(* IEC 61131-3 sources: TIA2AX/tests/V18/test_projects/expected/HW_2000482/6A1_AS10.2_AS11, 7 files *)

(* ---- HwIdentifiers.st ---- *)
TYPE
	HwIdentifiers : WORD
	(
		_6A1_AS10_2_AS11_Rail_0 :=	WORD#256,
		_6A1_AS10_2_AS11 :=	WORD#48,
		_6A1_AS10_2_AS11_Card_reader_writer_1 :=	WORD#51,
		_6A1_AS10_2_AS11_CPU_display_1 :=	WORD#54,
		_6A1_AS10_2_AS11_OPC_UA_1 :=	WORD#117,
		_6A1_AS10_2_AS11_PROFINET_interface_1 :=	WORD#64,
		_6A1_AS10_2_AS11_PROFINET_interface_1_Port_1 :=	WORD#65,
		_6A1_AS10_2_AS11_PROFINET_interface_1_Port_2 :=	WORD#66,
		_6A1_AS10_2_AS11_PROFINET_interface_2 :=	WORD#72,
		_6A1_AS10_2_AS11_PROFINET_interface_2_Port_1 :=	WORD#73,
		CPX_PneuOst_AS11_PN_IO_Interface :=	WORD#259,
		CPX_PneuOst_AS11_PN_IO_Interface_Port_1 :=	WORD#260,
		CPX_PneuOst_AS11_PN_IO_Interface_Port_2 :=	WORD#261,
		CPX_PneuOst_AS11_CPX :=	WORD#262,
		CPX_PneuOst_AS11_FB33_PNIO_Module_1 :=	WORD#263,
		CPX_PneuOst_AS11_MPA1S_VMPA1_FB_EMS_8_8DO_1 :=	WORD#264,
		CPX_PneuOst_AS11_MPA2S_VMPA2_FB_EMS_4_4DO_2 :=	WORD#265,
		CPX_PneuOst_AS11_MPA2S_VMPA2_FB_EMS_4_4DO_1 :=	WORD#266,
		CPX_PneuOst_AS11_MPA1S_VMPA1_FB_EMS_8_8DO_3 :=	WORD#267,
		CPX_PneuOst_AS11_MPA1S_VMPA1_FB_EMS_8_8DO_4 :=	WORD#268,
		CPX_PneuOst_AS11_MPA1G_VMPA1_FB_EMG_8_8DO_1 :=	WORD#269,
		_6A2_AS11_Rack_0 :=	WORD#273,
		_6A2_AS11 :=	WORD#274,
		_6A2_AS11_6A2_AS11 :=	WORD#275,
		_6A2_AS11_PROFINET_interface :=	WORD#276,
		_6A2_AS11_PROFINET_interface_Port_1 :=	WORD#278,
		_6A2_AS11_PROFINET_interface_Port_2 :=	WORD#277,
		_6A2_AS11_BA_2xRJ45 :=	WORD#278,
		_6A2_AS11_6A3 :=	WORD#279,
		_6A2_AS11_6A5 :=	WORD#280,
		_6A2_AS11_6A13 :=	WORD#281,
		_6A2_AS11_6A20 :=	WORD#282,
		_6A2_AS11_Server_module_1 :=	WORD#283,
		HousingReader_AS11_Rack :=	WORD#285,
		HousingReader_AS11 :=	WORD#286,
		HousingReader_AS11_Interface :=	WORD#287,
		HousingReader_AS11_Interface_Port_1 :=	WORD#288,
		HousingReader_AS11_SR_75X :=	WORD#289,
		HousingReader_AS11_Handshake_and_General_Error_Status_Bits_1 :=	WORD#290,
		HousingReader_AS11_BUSY_Status_Bits_1 :=	WORD#291,
		HousingReader_AS11_Completion_Status_Bits_1 :=	WORD#292,
		HousingReader_AS11_Error_Status_Bits_1 :=	WORD#293,
		HousingReader_AS11_Terminal_Status_Bits_1 :=	WORD#294,
		HousingReader_AS11_Unstable_Read_Status_Bits_1 :=	WORD#295,
		HousingReader_AS11_Matching_Level_and_Total_Evaluation_Grade_Status_1 :=	WORD#296,
		HousingReader_AS11_Operation_Result_Status_1 :=	WORD#297,
		HousingReader_AS11_Read_Data_128Byte_1 :=	WORD#298,
		HousingReader_AS11_Latch_and_Error_Clear_Control_Bits_1 :=	WORD#299,
		HousingReader_AS11_Operation_instruction_Control_Bits_1 :=	WORD#300,
		HousingReader_AS11_Completion_Clear_Control_Bits_1 :=	WORD#301,
		HousingReader_AS11_Parameter_Bank_Number_1 :=	WORD#302,
		HousingReader_AS11_User_Data_128Byte_1 :=	WORD#303,
		as13_lan_Rack :=	WORD#305,
		as13_lan :=	WORD#306,
		as13_lan_Interface :=	WORD#307,
		as13_lan_Interface_Port_1 :=	WORD#308,
		as13_lan_Interface_Port_2 :=	WORD#309,
		as13_lan_Communication :=	WORD#310,
		CPX_PneuOst_AS10_2_PN_IO_Interface :=	WORD#314,
		CPX_PneuOst_AS10_2_PN_IO_Interface_Port_1 :=	WORD#315,
		CPX_PneuOst_AS10_2_PN_IO_Interface_Port_2 :=	WORD#316,
		CPX_PneuOst_AS10_2_CPX :=	WORD#317,
		CPX_PneuOst_AS10_2_FB33_PNIO_Module_1 :=	WORD#318,
		CPX_PneuOst_AS10_2_MPA1S_VMPA1_FB_EMS_8_8DO_1 :=	WORD#319,
		CPX_PneuOst_AS10_2_MPA1S_VMPA1_FB_EMS_8_8DO_3 :=	WORD#320,
		CPX_PneuOst_AS10_2_MPA1S_VMPA1_FB_EMS_8_8DO_2 :=	WORD#321,
		CPX_PneuOst_AS10_2_MPA1G_VMPA1_FB_EMG_8_8DO_1 :=	WORD#322,
		FlashingReader_Rack :=	WORD#324,
		FlashingReader :=	WORD#325,
		FlashingReader_Interface :=	WORD#326,
		FlashingReader_Interface_Port_1 :=	WORD#327,
		FlashingReader_SR_75X :=	WORD#328,
		FlashingReader_Handshake_and_General_Error_Status_Bits_1 :=	WORD#329,
		FlashingReader_BUSY_Status_Bits_1 :=	WORD#330,
		FlashingReader_Completion_Status_Bits_1 :=	WORD#331,
		FlashingReader_Error_Status_Bits_1 :=	WORD#332,
		FlashingReader_Terminal_Status_Bits_1 :=	WORD#333,
		FlashingReader_Unstable_Read_Status_Bits_1 :=	WORD#334,
		FlashingReader_Matching_Level_and_Total_Evaluation_Grade_Status_1 :=	WORD#335,
		FlashingReader_Operation_Result_Status_1 :=	WORD#336,
		FlashingReader_Read_Data_128Byte_1 :=	WORD#337,
		FlashingReader_Latch_and_Error_Clear_Control_Bits_1 :=	WORD#338,
		FlashingReader_Operation_instruction_Control_Bits_1 :=	WORD#339,
		FlashingReader_Completion_Clear_Control_Bits_1 :=	WORD#340,
		FlashingReader_Parameter_Bank_Number_1 :=	WORD#341,
		FlashingReader_User_Data_128Byte_1 :=	WORD#342,
		AS10_2flashing_Interface1 :=	WORD#346,
		AS10_2flashing_Interface1_Port1 :=	WORD#347,
		AS10_2flashing_DF_Profinet_IO :=	WORD#348,
		AS10_2flashing_In_64_Byte_1 :=	WORD#349,
		AS10_2flashing_Out_64_Byte_1 :=	WORD#350,
		NONE:= WORD#0
	);
END_TYPE

(* ---- HwInputs.st ---- *)
TYPE
	HwInputs : STRUCT
		_6A2_AS11_6A3 AT %B0 : WORD;
		_6A2_AS11_6A13 AT %B19 : ARRAY[0..31] OF BYTE;
		HousingReader_AS11_Handshake_and_General_Error_Status_Bits_1 AT %B51 : BYTE;
		HousingReader_AS11_BUSY_Status_Bits_1 AT %B52 : BYTE;
		HousingReader_AS11_Completion_Status_Bits_1 AT %B53 : BYTE;
		HousingReader_AS11_Error_Status_Bits_1 AT %B54 : BYTE;
		HousingReader_AS11_Terminal_Status_Bits_1 AT %B55 : BYTE;
		HousingReader_AS11_Unstable_Read_Status_Bits_1 AT %B56 : BYTE;
		HousingReader_AS11_Matching_Level_and_Total_Evaluation_Grade_Status_1 AT %B57 : ARRAY[0..7] OF BYTE;
		HousingReader_AS11_Operation_Result_Status_1 AT %B65 : ARRAY[0..19] OF BYTE;
		HousingReader_AS11_Read_Data_128Byte_1 AT %B85 : ARRAY[0..135] OF BYTE;
		as13_lan_as13_lan AT %B221 : BYTE;
		FlashingReader_Handshake_and_General_Error_Status_Bits_1 AT %B222 : BYTE;
		FlashingReader_BUSY_Status_Bits_1 AT %B223 : BYTE;
		FlashingReader_Completion_Status_Bits_1 AT %B224 : BYTE;
		FlashingReader_Error_Status_Bits_1 AT %B225 : BYTE;
		FlashingReader_Terminal_Status_Bits_1 AT %B226 : BYTE;
		FlashingReader_Unstable_Read_Status_Bits_1 AT %B227 : BYTE;
		FlashingReader_Matching_Level_and_Total_Evaluation_Grade_Status_1 AT %B228 : ARRAY[0..7] OF BYTE;
		FlashingReader_Operation_Result_Status_1 AT %B236 : ARRAY[0..19] OF BYTE;
		FlashingReader_Read_Data_128Byte_1 AT %B256 : ARRAY[0..135] OF BYTE;
		AS10_2flashing_In_64_Byte_1 AT %B528 : ARRAY[0..63] OF BYTE;
	END_STRUCT;
END_TYPE

(* ---- HwOutputs.st ---- *)
TYPE
	HwOutputs : STRUCT
		CPX_PneuOst_AS11_MPA1S_VMPA1_FB_EMS_8_8DO_1 AT %B13 : BYTE;
		CPX_PneuOst_AS11_MPA2S_VMPA2_FB_EMS_4_4DO_2 AT %B183 : BYTE;
		CPX_PneuOst_AS11_MPA2S_VMPA2_FB_EMS_4_4DO_1 AT %B193 : BYTE;
		CPX_PneuOst_AS11_MPA1S_VMPA1_FB_EMS_8_8DO_3 AT %B184 : BYTE;
		CPX_PneuOst_AS11_MPA1S_VMPA1_FB_EMS_8_8DO_4 AT %B185 : BYTE;
		CPX_PneuOst_AS11_MPA1G_VMPA1_FB_EMG_8_8DO_1 AT %B186 : BYTE;
		_6A2_AS11_6A5 AT %B0 : WORD;
		_6A2_AS11_6A13 AT %B19 : ARRAY[0..31] OF BYTE;
		_6A2_AS11_6A20 AT %B328 : ARRAY[0..7] OF BYTE;
		HousingReader_AS11_Latch_and_Error_Clear_Control_Bits_1 AT %B6 : BYTE;
		HousingReader_AS11_Operation_instruction_Control_Bits_1 AT %B7 : BYTE;
		HousingReader_AS11_Completion_Clear_Control_Bits_1 AT %B12 : BYTE;
		HousingReader_AS11_Parameter_Bank_Number_1 AT %B51 : WORD;
		HousingReader_AS11_User_Data_128Byte_1 AT %B53 : ARRAY[0..129] OF BYTE;
		CPX_PneuOst_AS10_2_MPA1S_VMPA1_FB_EMS_8_8DO_1 AT %B188 : BYTE;
		CPX_PneuOst_AS10_2_MPA1S_VMPA1_FB_EMS_8_8DO_3 AT %B190 : BYTE;
		CPX_PneuOst_AS10_2_MPA1S_VMPA1_FB_EMS_8_8DO_2 AT %B194 : BYTE;
		CPX_PneuOst_AS10_2_MPA1G_VMPA1_FB_EMG_8_8DO_1 AT %B189 : BYTE;
		FlashingReader_Latch_and_Error_Clear_Control_Bits_1 AT %B191 : BYTE;
		FlashingReader_Operation_instruction_Control_Bits_1 AT %B192 : BYTE;
		FlashingReader_Completion_Clear_Control_Bits_1 AT %B195 : BYTE;
		FlashingReader_Parameter_Bank_Number_1 AT %B196 : WORD;
		FlashingReader_User_Data_128Byte_1 AT %B198 : ARRAY[0..129] OF BYTE;
		AS10_2flashing_Out_64_Byte_1 AT %B523 : ARRAY[0..63] OF BYTE;
	END_STRUCT;
END_TYPE

(* ---- PlcInputs.st ---- *)
TYPE
	PlcInputs : STRUCT
		_6A2_AS11_6A3 : WORD;
		_6A2_AS11_6A13 : ARRAY[0..31] OF BYTE;
		HousingReader_AS11_Handshake_and_General_Error_Status_Bits_1 : BYTE;
		HousingReader_AS11_BUSY_Status_Bits_1 : BYTE;
		HousingReader_AS11_Completion_Status_Bits_1 : BYTE;
		HousingReader_AS11_Error_Status_Bits_1 : BYTE;
		HousingReader_AS11_Terminal_Status_Bits_1 : BYTE;
		HousingReader_AS11_Unstable_Read_Status_Bits_1 : BYTE;
		HousingReader_AS11_Matching_Level_and_Total_Evaluation_Grade_Status_1 : ARRAY[0..7] OF BYTE;
		HousingReader_AS11_Operation_Result_Status_1 : ARRAY[0..19] OF BYTE;
		HousingReader_AS11_Read_Data_128Byte_1 : ARRAY[0..135] OF BYTE;
		as13_lan_as13_lan : BYTE;
		FlashingReader_Handshake_and_General_Error_Status_Bits_1 : BYTE;
		FlashingReader_BUSY_Status_Bits_1 : BYTE;
		FlashingReader_Completion_Status_Bits_1 : BYTE;
		FlashingReader_Error_Status_Bits_1 : BYTE;
		FlashingReader_Terminal_Status_Bits_1 : BYTE;
		FlashingReader_Unstable_Read_Status_Bits_1 : BYTE;
		FlashingReader_Matching_Level_and_Total_Evaluation_Grade_Status_1 : ARRAY[0..7] OF BYTE;
		FlashingReader_Operation_Result_Status_1 : ARRAY[0..19] OF BYTE;
		FlashingReader_Read_Data_128Byte_1 : ARRAY[0..135] OF BYTE;
		AS10_2flashing_In_64_Byte_1 : ARRAY[0..63] OF BYTE;
	END_STRUCT;
END_TYPE

(* ---- PlcOutputs.st ---- *)
TYPE
	PlcOutputs : STRUCT
		CPX_PneuOst_AS11_MPA1S_VMPA1_FB_EMS_8_8DO_1 : BYTE;
		CPX_PneuOst_AS11_MPA2S_VMPA2_FB_EMS_4_4DO_2 : BYTE;
		CPX_PneuOst_AS11_MPA2S_VMPA2_FB_EMS_4_4DO_1 : BYTE;
		CPX_PneuOst_AS11_MPA1S_VMPA1_FB_EMS_8_8DO_3 : BYTE;
		CPX_PneuOst_AS11_MPA1S_VMPA1_FB_EMS_8_8DO_4 : BYTE;
		CPX_PneuOst_AS11_MPA1G_VMPA1_FB_EMG_8_8DO_1 : BYTE;
		_6A2_AS11_6A5 : WORD;
		_6A2_AS11_6A13 : ARRAY[0..31] OF BYTE;
		_6A2_AS11_6A20 : ARRAY[0..7] OF BYTE;
		HousingReader_AS11_Latch_and_Error_Clear_Control_Bits_1 : BYTE;
		HousingReader_AS11_Operation_instruction_Control_Bits_1 : BYTE;
		HousingReader_AS11_Completion_Clear_Control_Bits_1 : BYTE;
		HousingReader_AS11_Parameter_Bank_Number_1 : WORD;
		HousingReader_AS11_User_Data_128Byte_1 : ARRAY[0..129] OF BYTE;
		CPX_PneuOst_AS10_2_MPA1S_VMPA1_FB_EMS_8_8DO_1 : BYTE;
		CPX_PneuOst_AS10_2_MPA1S_VMPA1_FB_EMS_8_8DO_3 : BYTE;
		CPX_PneuOst_AS10_2_MPA1S_VMPA1_FB_EMS_8_8DO_2 : BYTE;
		CPX_PneuOst_AS10_2_MPA1G_VMPA1_FB_EMG_8_8DO_1 : BYTE;
		FlashingReader_Latch_and_Error_Clear_Control_Bits_1 : BYTE;
		FlashingReader_Operation_instruction_Control_Bits_1 : BYTE;
		FlashingReader_Completion_Clear_Control_Bits_1 : BYTE;
		FlashingReader_Parameter_Bank_Number_1 : WORD;
		FlashingReader_User_Data_128Byte_1 : ARRAY[0..129] OF BYTE;
		AS10_2flashing_Out_64_Byte_1 : ARRAY[0..63] OF BYTE;
	END_STRUCT;
END_TYPE

(* ---- CopyInputs.st ---- *)
FUNCTION CopyInputs
	VAR_EXTERNAL
		HwInputs : HwInputs;
		PlcInputs : PlcInputs;
	END_VAR
	PlcInputs._6A2_AS11_6A3 := HwInputs._6A2_AS11_6A3;
	PlcInputs._6A2_AS11_6A13[0] := HwInputs._6A2_AS11_6A13[0];
	PlcInputs._6A2_AS11_6A13[1] := HwInputs._6A2_AS11_6A13[1];
	PlcInputs._6A2_AS11_6A13[2] := HwInputs._6A2_AS11_6A13[2];
	PlcInputs._6A2_AS11_6A13[3] := HwInputs._6A2_AS11_6A13[3];
	PlcInputs._6A2_AS11_6A13[4] := HwInputs._6A2_AS11_6A13[4];
	PlcInputs._6A2_AS11_6A13[5] := HwInputs._6A2_AS11_6A13[5];
	PlcInputs._6A2_AS11_6A13[6] := HwInputs._6A2_AS11_6A13[6];
	PlcInputs._6A2_AS11_6A13[7] := HwInputs._6A2_AS11_6A13[7];
	PlcInputs._6A2_AS11_6A13[8] := HwInputs._6A2_AS11_6A13[8];
	PlcInputs._6A2_AS11_6A13[9] := HwInputs._6A2_AS11_6A13[9];
	PlcInputs._6A2_AS11_6A13[10] := HwInputs._6A2_AS11_6A13[10];
	PlcInputs._6A2_AS11_6A13[11] := HwInputs._6A2_AS11_6A13[11];
	PlcInputs._6A2_AS11_6A13[12] := HwInputs._6A2_AS11_6A13[12];
	PlcInputs._6A2_AS11_6A13[13] := HwInputs._6A2_AS11_6A13[13];
	PlcInputs._6A2_AS11_6A13[14] := HwInputs._6A2_AS11_6A13[14];
	PlcInputs._6A2_AS11_6A13[15] := HwInputs._6A2_AS11_6A13[15];
	PlcInputs._6A2_AS11_6A13[16] := HwInputs._6A2_AS11_6A13[16];
	PlcInputs._6A2_AS11_6A13[17] := HwInputs._6A2_AS11_6A13[17];
	PlcInputs._6A2_AS11_6A13[18] := HwInputs._6A2_AS11_6A13[18];
	PlcInputs._6A2_AS11_6A13[19] := HwInputs._6A2_AS11_6A13[19];
	PlcInputs._6A2_AS11_6A13[20] := HwInputs._6A2_AS11_6A13[20];
	PlcInputs._6A2_AS11_6A13[21] := HwInputs._6A2_AS11_6A13[21];
	PlcInputs._6A2_AS11_6A13[22] := HwInputs._6A2_AS11_6A13[22];
	PlcInputs._6A2_AS11_6A13[23] := HwInputs._6A2_AS11_6A13[23];
	PlcInputs._6A2_AS11_6A13[24] := HwInputs._6A2_AS11_6A13[24];
	PlcInputs._6A2_AS11_6A13[25] := HwInputs._6A2_AS11_6A13[25];
	PlcInputs._6A2_AS11_6A13[26] := HwInputs._6A2_AS11_6A13[26];
	PlcInputs._6A2_AS11_6A13[27] := HwInputs._6A2_AS11_6A13[27];
	PlcInputs._6A2_AS11_6A13[28] := HwInputs._6A2_AS11_6A13[28];
	PlcInputs._6A2_AS11_6A13[29] := HwInputs._6A2_AS11_6A13[29];
	PlcInputs._6A2_AS11_6A13[30] := HwInputs._6A2_AS11_6A13[30];
	PlcInputs._6A2_AS11_6A13[31] := HwInputs._6A2_AS11_6A13[31];
	PlcInputs.HousingReader_AS11_Handshake_and_General_Error_Status_Bits_1 := HwInputs.HousingReader_AS11_Handshake_and_General_Error_Status_Bits_1;
	PlcInputs.HousingReader_AS11_BUSY_Status_Bits_1 := HwInputs.HousingReader_AS11_BUSY_Status_Bits_1;
	PlcInputs.HousingReader_AS11_Completion_Status_Bits_1 := HwInputs.HousingReader_AS11_Completion_Status_Bits_1;
	PlcInputs.HousingReader_AS11_Error_Status_Bits_1 := HwInputs.HousingReader_AS11_Error_Status_Bits_1;
	PlcInputs.HousingReader_AS11_Terminal_Status_Bits_1 := HwInputs.HousingReader_AS11_Terminal_Status_Bits_1;
	PlcInputs.HousingReader_AS11_Unstable_Read_Status_Bits_1 := HwInputs.HousingReader_AS11_Unstable_Read_Status_Bits_1;
	PlcInputs.HousingReader_AS11_Matching_Level_and_Total_Evaluation_Grade_Status_1[0] := HwInputs.HousingReader_AS11_Matching_Level_and_Total_Evaluation_Grade_Status_1[0];
	PlcInputs.HousingReader_AS11_Matching_Level_and_Total_Evaluation_Grade_Status_1[1] := HwInputs.HousingReader_AS11_Matching_Level_and_Total_Evaluation_Grade_Status_1[1];
	PlcInputs.HousingReader_AS11_Matching_Level_and_Total_Evaluation_Grade_Status_1[2] := HwInputs.HousingReader_AS11_Matching_Level_and_Total_Evaluation_Grade_Status_1[2];
	PlcInputs.HousingReader_AS11_Matching_Level_and_Total_Evaluation_Grade_Status_1[3] := HwInputs.HousingReader_AS11_Matching_Level_and_Total_Evaluation_Grade_Status_1[3];
	PlcInputs.HousingReader_AS11_Matching_Level_and_Total_Evaluation_Grade_Status_1[4] := HwInputs.HousingReader_AS11_Matching_Level_and_Total_Evaluation_Grade_Status_1[4];
	PlcInputs.HousingReader_AS11_Matching_Level_and_Total_Evaluation_Grade_Status_1[5] := HwInputs.HousingReader_AS11_Matching_Level_and_Total_Evaluation_Grade_Status_1[5];
	PlcInputs.HousingReader_AS11_Matching_Level_and_Total_Evaluation_Grade_Status_1[6] := HwInputs.HousingReader_AS11_Matching_Level_and_Total_Evaluation_Grade_Status_1[6];
	PlcInputs.HousingReader_AS11_Matching_Level_and_Total_Evaluation_Grade_Status_1[7] := HwInputs.HousingReader_AS11_Matching_Level_and_Total_Evaluation_Grade_Status_1[7];
	PlcInputs.HousingReader_AS11_Operation_Result_Status_1[0] := HwInputs.HousingReader_AS11_Operation_Result_Status_1[0];
	PlcInputs.HousingReader_AS11_Operation_Result_Status_1[1] := HwInputs.HousingReader_AS11_Operation_Result_Status_1[1];
	PlcInputs.HousingReader_AS11_Operation_Result_Status_1[2] := HwInputs.HousingReader_AS11_Operation_Result_Status_1[2];
	PlcInputs.HousingReader_AS11_Operation_Result_Status_1[3] := HwInputs.HousingReader_AS11_Operation_Result_Status_1[3];
	PlcInputs.HousingReader_AS11_Operation_Result_Status_1[4] := HwInputs.HousingReader_AS11_Operation_Result_Status_1[4];
	PlcInputs.HousingReader_AS11_Operation_Result_Status_1[5] := HwInputs.HousingReader_AS11_Operation_Result_Status_1[5];
	PlcInputs.HousingReader_AS11_Operation_Result_Status_1[6] := HwInputs.HousingReader_AS11_Operation_Result_Status_1[6];
	PlcInputs.HousingReader_AS11_Operation_Result_Status_1[7] := HwInputs.HousingReader_AS11_Operation_Result_Status_1[7];
	PlcInputs.HousingReader_AS11_Operation_Result_Status_1[8] := HwInputs.HousingReader_AS11_Operation_Result_Status_1[8];
	PlcInputs.HousingReader_AS11_Operation_Result_Status_1[9] := HwInputs.HousingReader_AS11_Operation_Result_Status_1[9];
	PlcInputs.HousingReader_AS11_Operation_Result_Status_1[10] := HwInputs.HousingReader_AS11_Operation_Result_Status_1[10];
	PlcInputs.HousingReader_AS11_Operation_Result_Status_1[11] := HwInputs.HousingReader_AS11_Operation_Result_Status_1[11];
	PlcInputs.HousingReader_AS11_Operation_Result_Status_1[12] := HwInputs.HousingReader_AS11_Operation_Result_Status_1[12];
	PlcInputs.HousingReader_AS11_Operation_Result_Status_1[13] := HwInputs.HousingReader_AS11_Operation_Result_Status_1[13];
	PlcInputs.HousingReader_AS11_Operation_Result_Status_1[14] := HwInputs.HousingReader_AS11_Operation_Result_Status_1[14];
	PlcInputs.HousingReader_AS11_Operation_Result_Status_1[15] := HwInputs.HousingReader_AS11_Operation_Result_Status_1[15];
	PlcInputs.HousingReader_AS11_Operation_Result_Status_1[16] := HwInputs.HousingReader_AS11_Operation_Result_Status_1[16];
	PlcInputs.HousingReader_AS11_Operation_Result_Status_1[17] := HwInputs.HousingReader_AS11_Operation_Result_Status_1[17];
	PlcInputs.HousingReader_AS11_Operation_Result_Status_1[18] := HwInputs.HousingReader_AS11_Operation_Result_Status_1[18];
	PlcInputs.HousingReader_AS11_Operation_Result_Status_1[19] := HwInputs.HousingReader_AS11_Operation_Result_Status_1[19];
	PlcInputs.HousingReader_AS11_Read_Data_128Byte_1[0] := HwInputs.HousingReader_AS11_Read_Data_128Byte_1[0];
	PlcInputs.HousingReader_AS11_Read_Data_128Byte_1[1] := HwInputs.HousingReader_AS11_Read_Data_128Byte_1[1];
	PlcInputs.HousingReader_AS11_Read_Data_128Byte_1[2] := HwInputs.HousingReader_AS11_Read_Data_128Byte_1[2];
	PlcInputs.HousingReader_AS11_Read_Data_128Byte_1[3] := HwInputs.HousingReader_AS11_Read_Data_128Byte_1[3];
	PlcInputs.HousingReader_AS11_Read_Data_128Byte_1[4] := HwInputs.HousingReader_AS11_Read_Data_128Byte_1[4];
	PlcInputs.HousingReader_AS11_Read_Data_128Byte_1[5] := HwInputs.HousingReader_AS11_Read_Data_128Byte_1[5];
	PlcInputs.HousingReader_AS11_Read_Data_128Byte_1[6] := HwInputs.HousingReader_AS11_Read_Data_128Byte_1[6];
	PlcInputs.HousingReader_AS11_Read_Data_128Byte_1[7] := HwInputs.HousingReader_AS11_Read_Data_128Byte_1[7];
	PlcInputs.HousingReader_AS11_Read_Data_128Byte_1[8] := HwInputs.HousingReader_AS11_Read_Data_128Byte_1[8];
	PlcInputs.HousingReader_AS11_Read_Data_128Byte_1[9] := HwInputs.HousingReader_AS11_Read_Data_128Byte_1[9];
	PlcInputs.HousingReader_AS11_Read_Data_128Byte_1[10] := HwInputs.HousingReader_AS11_Read_Data_128Byte_1[10];
	PlcInputs.HousingReader_AS11_Read_Data_128Byte_1[11] := HwInputs.HousingReader_AS11_Read_Data_128Byte_1[11];
	PlcInputs.HousingReader_AS11_Read_Data_128Byte_1[12] := HwInputs.HousingReader_AS11_Read_Data_128Byte_1[12];
	PlcInputs.HousingReader_AS11_Read_Data_128Byte_1[13] := HwInputs.HousingReader_AS11_Read_Data_128Byte_1[13];
	PlcInputs.HousingReader_AS11_Read_Data_128Byte_1[14] := HwInputs.HousingReader_AS11_Read_Data_128Byte_1[14];
	PlcInputs.HousingReader_AS11_Read_Data_128Byte_1[15] := HwInputs.HousingReader_AS11_Read_Data_128Byte_1[15];
	PlcInputs.HousingReader_AS11_Read_Data_128Byte_1[16] := HwInputs.HousingReader_AS11_Read_Data_128Byte_1[16];
	PlcInputs.HousingReader_AS11_Read_Data_128Byte_1[17] := HwInputs.HousingReader_AS11_Read_Data_128Byte_1[17];
	PlcInputs.HousingReader_AS11_Read_Data_128Byte_1[18] := HwInputs.HousingReader_AS11_Read_Data_128Byte_1[18];
	PlcInputs.HousingReader_AS11_Read_Data_128Byte_1[19] := HwInputs.HousingReader_AS11_Read_Data_128Byte_1[19];
	PlcInputs.HousingReader_AS11_Read_Data_128Byte_1[20] := HwInputs.HousingReader_AS11_Read_Data_128Byte_1[20];
	PlcInputs.HousingReader_AS11_Read_Data_128Byte_1[21] := HwInputs.HousingReader_AS11_Read_Data_128Byte_1[21];
	PlcInputs.HousingReader_AS11_Read_Data_128Byte_1[22] := HwInputs.HousingReader_AS11_Read_Data_128Byte_1[22];
	PlcInputs.HousingReader_AS11_Read_Data_128Byte_1[23] := HwInputs.HousingReader_AS11_Read_Data_128Byte_1[23];
	PlcInputs.HousingReader_AS11_Read_Data_128Byte_1[24] := HwInputs.HousingReader_AS11_Read_Data_128Byte_1[24];
	PlcInputs.HousingReader_AS11_Read_Data_128Byte_1[25] := HwInputs.HousingReader_AS11_Read_Data_128Byte_1[25];
	PlcInputs.HousingReader_AS11_Read_Data_128Byte_1[26] := HwInputs.HousingReader_AS11_Read_Data_128Byte_1[26];
	PlcInputs.HousingReader_AS11_Read_Data_128Byte_1[27] := HwInputs.HousingReader_AS11_Read_Data_128Byte_1[27];
	PlcInputs.HousingReader_AS11_Read_Data_128Byte_1[28] := HwInputs.HousingReader_AS11_Read_Data_128Byte_1[28];
	PlcInputs.HousingReader_AS11_Read_Data_128Byte_1[29] := HwInputs.HousingReader_AS11_Read_Data_128Byte_1[29];
	PlcInputs.HousingReader_AS11_Read_Data_128Byte_1[30] := HwInputs.HousingReader_AS11_Read_Data_128Byte_1[30];
	PlcInputs.HousingReader_AS11_Read_Data_128Byte_1[31] := HwInputs.HousingReader_AS11_Read_Data_128Byte_1[31];
	PlcInputs.HousingReader_AS11_Read_Data_128Byte_1[32] := HwInputs.HousingReader_AS11_Read_Data_128Byte_1[32];
	PlcInputs.HousingReader_AS11_Read_Data_128Byte_1[33] := HwInputs.HousingReader_AS11_Read_Data_128Byte_1[33];
	PlcInputs.HousingReader_AS11_Read_Data_128Byte_1[34] := HwInputs.HousingReader_AS11_Read_Data_128Byte_1[34];
	PlcInputs.HousingReader_AS11_Read_Data_128Byte_1[35] := HwInputs.HousingReader_AS11_Read_Data_128Byte_1[35];
	PlcInputs.HousingReader_AS11_Read_Data_128Byte_1[36] := HwInputs.HousingReader_AS11_Read_Data_128Byte_1[36];
	PlcInputs.HousingReader_AS11_Read_Data_128Byte_1[37] := HwInputs.HousingReader_AS11_Read_Data_128Byte_1[37];
	PlcInputs.HousingReader_AS11_Read_Data_128Byte_1[38] := HwInputs.HousingReader_AS11_Read_Data_128Byte_1[38];
	PlcInputs.HousingReader_AS11_Read_Data_128Byte_1[39] := HwInputs.HousingReader_AS11_Read_Data_128Byte_1[39];
	PlcInputs.HousingReader_AS11_Read_Data_128Byte_1[40] := HwInputs.HousingReader_AS11_Read_Data_128Byte_1[40];
	PlcInputs.HousingReader_AS11_Read_Data_128Byte_1[41] := HwInputs.HousingReader_AS11_Read_Data_128Byte_1[41];
	PlcInputs.HousingReader_AS11_Read_Data_128Byte_1[42] := HwInputs.HousingReader_AS11_Read_Data_128Byte_1[42];
	PlcInputs.HousingReader_AS11_Read_Data_128Byte_1[43] := HwInputs.HousingReader_AS11_Read_Data_128Byte_1[43];
	PlcInputs.HousingReader_AS11_Read_Data_128Byte_1[44] := HwInputs.HousingReader_AS11_Read_Data_128Byte_1[44];
	PlcInputs.HousingReader_AS11_Read_Data_128Byte_1[45] := HwInputs.HousingReader_AS11_Read_Data_128Byte_1[45];
	PlcInputs.HousingReader_AS11_Read_Data_128Byte_1[46] := HwInputs.HousingReader_AS11_Read_Data_128Byte_1[46];
	PlcInputs.HousingReader_AS11_Read_Data_128Byte_1[47] := HwInputs.HousingReader_AS11_Read_Data_128Byte_1[47];
	PlcInputs.HousingReader_AS11_Read_Data_128Byte_1[48] := HwInputs.HousingReader_AS11_Read_Data_128Byte_1[48];
	PlcInputs.HousingReader_AS11_Read_Data_128Byte_1[49] := HwInputs.HousingReader_AS11_Read_Data_128Byte_1[49];
	PlcInputs.HousingReader_AS11_Read_Data_128Byte_1[50] := HwInputs.HousingReader_AS11_Read_Data_128Byte_1[50];
	PlcInputs.HousingReader_AS11_Read_Data_128Byte_1[51] := HwInputs.HousingReader_AS11_Read_Data_128Byte_1[51];
	PlcInputs.HousingReader_AS11_Read_Data_128Byte_1[52] := HwInputs.HousingReader_AS11_Read_Data_128Byte_1[52];
	PlcInputs.HousingReader_AS11_Read_Data_128Byte_1[53] := HwInputs.HousingReader_AS11_Read_Data_128Byte_1[53];
	PlcInputs.HousingReader_AS11_Read_Data_128Byte_1[54] := HwInputs.HousingReader_AS11_Read_Data_128Byte_1[54];
	PlcInputs.HousingReader_AS11_Read_Data_128Byte_1[55] := HwInputs.HousingReader_AS11_Read_Data_128Byte_1[55];
	PlcInputs.HousingReader_AS11_Read_Data_128Byte_1[56] := HwInputs.HousingReader_AS11_Read_Data_128Byte_1[56];
	PlcInputs.HousingReader_AS11_Read_Data_128Byte_1[57] := HwInputs.HousingReader_AS11_Read_Data_128Byte_1[57];
	PlcInputs.HousingReader_AS11_Read_Data_128Byte_1[58] := HwInputs.HousingReader_AS11_Read_Data_128Byte_1[58];
	PlcInputs.HousingReader_AS11_Read_Data_128Byte_1[59] := HwInputs.HousingReader_AS11_Read_Data_128Byte_1[59];
	PlcInputs.HousingReader_AS11_Read_Data_128Byte_1[60] := HwInputs.HousingReader_AS11_Read_Data_128Byte_1[60];
	PlcInputs.HousingReader_AS11_Read_Data_128Byte_1[61] := HwInputs.HousingReader_AS11_Read_Data_128Byte_1[61];
	PlcInputs.HousingReader_AS11_Read_Data_128Byte_1[62] := HwInputs.HousingReader_AS11_Read_Data_128Byte_1[62];
	PlcInputs.HousingReader_AS11_Read_Data_128Byte_1[63] := HwInputs.HousingReader_AS11_Read_Data_128Byte_1[63];
	PlcInputs.HousingReader_AS11_Read_Data_128Byte_1[64] := HwInputs.HousingReader_AS11_Read_Data_128Byte_1[64];
	PlcInputs.HousingReader_AS11_Read_Data_128Byte_1[65] := HwInputs.HousingReader_AS11_Read_Data_128Byte_1[65];
	PlcInputs.HousingReader_AS11_Read_Data_128Byte_1[66] := HwInputs.HousingReader_AS11_Read_Data_128Byte_1[66];
	PlcInputs.HousingReader_AS11_Read_Data_128Byte_1[67] := HwInputs.HousingReader_AS11_Read_Data_128Byte_1[67];
	PlcInputs.HousingReader_AS11_Read_Data_128Byte_1[68] := HwInputs.HousingReader_AS11_Read_Data_128Byte_1[68];
	PlcInputs.HousingReader_AS11_Read_Data_128Byte_1[69] := HwInputs.HousingReader_AS11_Read_Data_128Byte_1[69];
	PlcInputs.HousingReader_AS11_Read_Data_128Byte_1[70] := HwInputs.HousingReader_AS11_Read_Data_128Byte_1[70];
	PlcInputs.HousingReader_AS11_Read_Data_128Byte_1[71] := HwInputs.HousingReader_AS11_Read_Data_128Byte_1[71];
	PlcInputs.HousingReader_AS11_Read_Data_128Byte_1[72] := HwInputs.HousingReader_AS11_Read_Data_128Byte_1[72];
	PlcInputs.HousingReader_AS11_Read_Data_128Byte_1[73] := HwInputs.HousingReader_AS11_Read_Data_128Byte_1[73];
	PlcInputs.HousingReader_AS11_Read_Data_128Byte_1[74] := HwInputs.HousingReader_AS11_Read_Data_128Byte_1[74];
	PlcInputs.HousingReader_AS11_Read_Data_128Byte_1[75] := HwInputs.HousingReader_AS11_Read_Data_128Byte_1[75];
	PlcInputs.HousingReader_AS11_Read_Data_128Byte_1[76] := HwInputs.HousingReader_AS11_Read_Data_128Byte_1[76];
	PlcInputs.HousingReader_AS11_Read_Data_128Byte_1[77] := HwInputs.HousingReader_AS11_Read_Data_128Byte_1[77];
	PlcInputs.HousingReader_AS11_Read_Data_128Byte_1[78] := HwInputs.HousingReader_AS11_Read_Data_128Byte_1[78];
	PlcInputs.HousingReader_AS11_Read_Data_128Byte_1[79] := HwInputs.HousingReader_AS11_Read_Data_128Byte_1[79];
	PlcInputs.HousingReader_AS11_Read_Data_128Byte_1[80] := HwInputs.HousingReader_AS11_Read_Data_128Byte_1[80];
	PlcInputs.HousingReader_AS11_Read_Data_128Byte_1[81] := HwInputs.HousingReader_AS11_Read_Data_128Byte_1[81];
	PlcInputs.HousingReader_AS11_Read_Data_128Byte_1[82] := HwInputs.HousingReader_AS11_Read_Data_128Byte_1[82];
	PlcInputs.HousingReader_AS11_Read_Data_128Byte_1[83] := HwInputs.HousingReader_AS11_Read_Data_128Byte_1[83];
	PlcInputs.HousingReader_AS11_Read_Data_128Byte_1[84] := HwInputs.HousingReader_AS11_Read_Data_128Byte_1[84];
	PlcInputs.HousingReader_AS11_Read_Data_128Byte_1[85] := HwInputs.HousingReader_AS11_Read_Data_128Byte_1[85];
	PlcInputs.HousingReader_AS11_Read_Data_128Byte_1[86] := HwInputs.HousingReader_AS11_Read_Data_128Byte_1[86];
	PlcInputs.HousingReader_AS11_Read_Data_128Byte_1[87] := HwInputs.HousingReader_AS11_Read_Data_128Byte_1[87];
	PlcInputs.HousingReader_AS11_Read_Data_128Byte_1[88] := HwInputs.HousingReader_AS11_Read_Data_128Byte_1[88];
	PlcInputs.HousingReader_AS11_Read_Data_128Byte_1[89] := HwInputs.HousingReader_AS11_Read_Data_128Byte_1[89];
	PlcInputs.HousingReader_AS11_Read_Data_128Byte_1[90] := HwInputs.HousingReader_AS11_Read_Data_128Byte_1[90];
	PlcInputs.HousingReader_AS11_Read_Data_128Byte_1[91] := HwInputs.HousingReader_AS11_Read_Data_128Byte_1[91];
	PlcInputs.HousingReader_AS11_Read_Data_128Byte_1[92] := HwInputs.HousingReader_AS11_Read_Data_128Byte_1[92];
	PlcInputs.HousingReader_AS11_Read_Data_128Byte_1[93] := HwInputs.HousingReader_AS11_Read_Data_128Byte_1[93];
	PlcInputs.HousingReader_AS11_Read_Data_128Byte_1[94] := HwInputs.HousingReader_AS11_Read_Data_128Byte_1[94];
	PlcInputs.HousingReader_AS11_Read_Data_128Byte_1[95] := HwInputs.HousingReader_AS11_Read_Data_128Byte_1[95];
	PlcInputs.HousingReader_AS11_Read_Data_128Byte_1[96] := HwInputs.HousingReader_AS11_Read_Data_128Byte_1[96];
	PlcInputs.HousingReader_AS11_Read_Data_128Byte_1[97] := HwInputs.HousingReader_AS11_Read_Data_128Byte_1[97];
	PlcInputs.HousingReader_AS11_Read_Data_128Byte_1[98] := HwInputs.HousingReader_AS11_Read_Data_128Byte_1[98];
	PlcInputs.HousingReader_AS11_Read_Data_128Byte_1[99] := HwInputs.HousingReader_AS11_Read_Data_128Byte_1[99];
	PlcInputs.HousingReader_AS11_Read_Data_128Byte_1[100] := HwInputs.HousingReader_AS11_Read_Data_128Byte_1[100];
	PlcInputs.HousingReader_AS11_Read_Data_128Byte_1[101] := HwInputs.HousingReader_AS11_Read_Data_128Byte_1[101];
	PlcInputs.HousingReader_AS11_Read_Data_128Byte_1[102] := HwInputs.HousingReader_AS11_Read_Data_128Byte_1[102];
	PlcInputs.HousingReader_AS11_Read_Data_128Byte_1[103] := HwInputs.HousingReader_AS11_Read_Data_128Byte_1[103];
	PlcInputs.HousingReader_AS11_Read_Data_128Byte_1[104] := HwInputs.HousingReader_AS11_Read_Data_128Byte_1[104];
	PlcInputs.HousingReader_AS11_Read_Data_128Byte_1[105] := HwInputs.HousingReader_AS11_Read_Data_128Byte_1[105];
	PlcInputs.HousingReader_AS11_Read_Data_128Byte_1[106] := HwInputs.HousingReader_AS11_Read_Data_128Byte_1[106];
	PlcInputs.HousingReader_AS11_Read_Data_128Byte_1[107] := HwInputs.HousingReader_AS11_Read_Data_128Byte_1[107];
	PlcInputs.HousingReader_AS11_Read_Data_128Byte_1[108] := HwInputs.HousingReader_AS11_Read_Data_128Byte_1[108];
	PlcInputs.HousingReader_AS11_Read_Data_128Byte_1[109] := HwInputs.HousingReader_AS11_Read_Data_128Byte_1[109];
	PlcInputs.HousingReader_AS11_Read_Data_128Byte_1[110] := HwInputs.HousingReader_AS11_Read_Data_128Byte_1[110];
	PlcInputs.HousingReader_AS11_Read_Data_128Byte_1[111] := HwInputs.HousingReader_AS11_Read_Data_128Byte_1[111];
	PlcInputs.HousingReader_AS11_Read_Data_128Byte_1[112] := HwInputs.HousingReader_AS11_Read_Data_128Byte_1[112];
	PlcInputs.HousingReader_AS11_Read_Data_128Byte_1[113] := HwInputs.HousingReader_AS11_Read_Data_128Byte_1[113];
	PlcInputs.HousingReader_AS11_Read_Data_128Byte_1[114] := HwInputs.HousingReader_AS11_Read_Data_128Byte_1[114];
	PlcInputs.HousingReader_AS11_Read_Data_128Byte_1[115] := HwInputs.HousingReader_AS11_Read_Data_128Byte_1[115];
	PlcInputs.HousingReader_AS11_Read_Data_128Byte_1[116] := HwInputs.HousingReader_AS11_Read_Data_128Byte_1[116];
	PlcInputs.HousingReader_AS11_Read_Data_128Byte_1[117] := HwInputs.HousingReader_AS11_Read_Data_128Byte_1[117];
	PlcInputs.HousingReader_AS11_Read_Data_128Byte_1[118] := HwInputs.HousingReader_AS11_Read_Data_128Byte_1[118];
	PlcInputs.HousingReader_AS11_Read_Data_128Byte_1[119] := HwInputs.HousingReader_AS11_Read_Data_128Byte_1[119];
	PlcInputs.HousingReader_AS11_Read_Data_128Byte_1[120] := HwInputs.HousingReader_AS11_Read_Data_128Byte_1[120];
	PlcInputs.HousingReader_AS11_Read_Data_128Byte_1[121] := HwInputs.HousingReader_AS11_Read_Data_128Byte_1[121];
	PlcInputs.HousingReader_AS11_Read_Data_128Byte_1[122] := HwInputs.HousingReader_AS11_Read_Data_128Byte_1[122];
	PlcInputs.HousingReader_AS11_Read_Data_128Byte_1[123] := HwInputs.HousingReader_AS11_Read_Data_128Byte_1[123];
	PlcInputs.HousingReader_AS11_Read_Data_128Byte_1[124] := HwInputs.HousingReader_AS11_Read_Data_128Byte_1[124];
	PlcInputs.HousingReader_AS11_Read_Data_128Byte_1[125] := HwInputs.HousingReader_AS11_Read_Data_128Byte_1[125];
	PlcInputs.HousingReader_AS11_Read_Data_128Byte_1[126] := HwInputs.HousingReader_AS11_Read_Data_128Byte_1[126];
	PlcInputs.HousingReader_AS11_Read_Data_128Byte_1[127] := HwInputs.HousingReader_AS11_Read_Data_128Byte_1[127];
	PlcInputs.HousingReader_AS11_Read_Data_128Byte_1[128] := HwInputs.HousingReader_AS11_Read_Data_128Byte_1[128];
	PlcInputs.HousingReader_AS11_Read_Data_128Byte_1[129] := HwInputs.HousingReader_AS11_Read_Data_128Byte_1[129];
	PlcInputs.HousingReader_AS11_Read_Data_128Byte_1[130] := HwInputs.HousingReader_AS11_Read_Data_128Byte_1[130];
	PlcInputs.HousingReader_AS11_Read_Data_128Byte_1[131] := HwInputs.HousingReader_AS11_Read_Data_128Byte_1[131];
	PlcInputs.HousingReader_AS11_Read_Data_128Byte_1[132] := HwInputs.HousingReader_AS11_Read_Data_128Byte_1[132];
	PlcInputs.HousingReader_AS11_Read_Data_128Byte_1[133] := HwInputs.HousingReader_AS11_Read_Data_128Byte_1[133];
	PlcInputs.HousingReader_AS11_Read_Data_128Byte_1[134] := HwInputs.HousingReader_AS11_Read_Data_128Byte_1[134];
	PlcInputs.HousingReader_AS11_Read_Data_128Byte_1[135] := HwInputs.HousingReader_AS11_Read_Data_128Byte_1[135];
	PlcInputs.as13_lan_as13_lan := HwInputs.as13_lan_as13_lan;
	PlcInputs.FlashingReader_Handshake_and_General_Error_Status_Bits_1 := HwInputs.FlashingReader_Handshake_and_General_Error_Status_Bits_1;
	PlcInputs.FlashingReader_BUSY_Status_Bits_1 := HwInputs.FlashingReader_BUSY_Status_Bits_1;
	PlcInputs.FlashingReader_Completion_Status_Bits_1 := HwInputs.FlashingReader_Completion_Status_Bits_1;
	PlcInputs.FlashingReader_Error_Status_Bits_1 := HwInputs.FlashingReader_Error_Status_Bits_1;
	PlcInputs.FlashingReader_Terminal_Status_Bits_1 := HwInputs.FlashingReader_Terminal_Status_Bits_1;
	PlcInputs.FlashingReader_Unstable_Read_Status_Bits_1 := HwInputs.FlashingReader_Unstable_Read_Status_Bits_1;
	PlcInputs.FlashingReader_Matching_Level_and_Total_Evaluation_Grade_Status_1[0] := HwInputs.FlashingReader_Matching_Level_and_Total_Evaluation_Grade_Status_1[0];
	PlcInputs.FlashingReader_Matching_Level_and_Total_Evaluation_Grade_Status_1[1] := HwInputs.FlashingReader_Matching_Level_and_Total_Evaluation_Grade_Status_1[1];
	PlcInputs.FlashingReader_Matching_Level_and_Total_Evaluation_Grade_Status_1[2] := HwInputs.FlashingReader_Matching_Level_and_Total_Evaluation_Grade_Status_1[2];
	PlcInputs.FlashingReader_Matching_Level_and_Total_Evaluation_Grade_Status_1[3] := HwInputs.FlashingReader_Matching_Level_and_Total_Evaluation_Grade_Status_1[3];
	PlcInputs.FlashingReader_Matching_Level_and_Total_Evaluation_Grade_Status_1[4] := HwInputs.FlashingReader_Matching_Level_and_Total_Evaluation_Grade_Status_1[4];
	PlcInputs.FlashingReader_Matching_Level_and_Total_Evaluation_Grade_Status_1[5] := HwInputs.FlashingReader_Matching_Level_and_Total_Evaluation_Grade_Status_1[5];
	PlcInputs.FlashingReader_Matching_Level_and_Total_Evaluation_Grade_Status_1[6] := HwInputs.FlashingReader_Matching_Level_and_Total_Evaluation_Grade_Status_1[6];
	PlcInputs.FlashingReader_Matching_Level_and_Total_Evaluation_Grade_Status_1[7] := HwInputs.FlashingReader_Matching_Level_and_Total_Evaluation_Grade_Status_1[7];
	PlcInputs.FlashingReader_Operation_Result_Status_1[0] := HwInputs.FlashingReader_Operation_Result_Status_1[0];
	PlcInputs.FlashingReader_Operation_Result_Status_1[1] := HwInputs.FlashingReader_Operation_Result_Status_1[1];
	PlcInputs.FlashingReader_Operation_Result_Status_1[2] := HwInputs.FlashingReader_Operation_Result_Status_1[2];
	PlcInputs.FlashingReader_Operation_Result_Status_1[3] := HwInputs.FlashingReader_Operation_Result_Status_1[3];
	PlcInputs.FlashingReader_Operation_Result_Status_1[4] := HwInputs.FlashingReader_Operation_Result_Status_1[4];
	PlcInputs.FlashingReader_Operation_Result_Status_1[5] := HwInputs.FlashingReader_Operation_Result_Status_1[5];
	PlcInputs.FlashingReader_Operation_Result_Status_1[6] := HwInputs.FlashingReader_Operation_Result_Status_1[6];
	PlcInputs.FlashingReader_Operation_Result_Status_1[7] := HwInputs.FlashingReader_Operation_Result_Status_1[7];
	PlcInputs.FlashingReader_Operation_Result_Status_1[8] := HwInputs.FlashingReader_Operation_Result_Status_1[8];
	PlcInputs.FlashingReader_Operation_Result_Status_1[9] := HwInputs.FlashingReader_Operation_Result_Status_1[9];
	PlcInputs.FlashingReader_Operation_Result_Status_1[10] := HwInputs.FlashingReader_Operation_Result_Status_1[10];
	PlcInputs.FlashingReader_Operation_Result_Status_1[11] := HwInputs.FlashingReader_Operation_Result_Status_1[11];
	PlcInputs.FlashingReader_Operation_Result_Status_1[12] := HwInputs.FlashingReader_Operation_Result_Status_1[12];
	PlcInputs.FlashingReader_Operation_Result_Status_1[13] := HwInputs.FlashingReader_Operation_Result_Status_1[13];
	PlcInputs.FlashingReader_Operation_Result_Status_1[14] := HwInputs.FlashingReader_Operation_Result_Status_1[14];
	PlcInputs.FlashingReader_Operation_Result_Status_1[15] := HwInputs.FlashingReader_Operation_Result_Status_1[15];
	PlcInputs.FlashingReader_Operation_Result_Status_1[16] := HwInputs.FlashingReader_Operation_Result_Status_1[16];
	PlcInputs.FlashingReader_Operation_Result_Status_1[17] := HwInputs.FlashingReader_Operation_Result_Status_1[17];
	PlcInputs.FlashingReader_Operation_Result_Status_1[18] := HwInputs.FlashingReader_Operation_Result_Status_1[18];
	PlcInputs.FlashingReader_Operation_Result_Status_1[19] := HwInputs.FlashingReader_Operation_Result_Status_1[19];
	PlcInputs.FlashingReader_Read_Data_128Byte_1[0] := HwInputs.FlashingReader_Read_Data_128Byte_1[0];
	PlcInputs.FlashingReader_Read_Data_128Byte_1[1] := HwInputs.FlashingReader_Read_Data_128Byte_1[1];
	PlcInputs.FlashingReader_Read_Data_128Byte_1[2] := HwInputs.FlashingReader_Read_Data_128Byte_1[2];
	PlcInputs.FlashingReader_Read_Data_128Byte_1[3] := HwInputs.FlashingReader_Read_Data_128Byte_1[3];
	PlcInputs.FlashingReader_Read_Data_128Byte_1[4] := HwInputs.FlashingReader_Read_Data_128Byte_1[4];
	PlcInputs.FlashingReader_Read_Data_128Byte_1[5] := HwInputs.FlashingReader_Read_Data_128Byte_1[5];
	PlcInputs.FlashingReader_Read_Data_128Byte_1[6] := HwInputs.FlashingReader_Read_Data_128Byte_1[6];
	PlcInputs.FlashingReader_Read_Data_128Byte_1[7] := HwInputs.FlashingReader_Read_Data_128Byte_1[7];
	PlcInputs.FlashingReader_Read_Data_128Byte_1[8] := HwInputs.FlashingReader_Read_Data_128Byte_1[8];
	PlcInputs.FlashingReader_Read_Data_128Byte_1[9] := HwInputs.FlashingReader_Read_Data_128Byte_1[9];
	PlcInputs.FlashingReader_Read_Data_128Byte_1[10] := HwInputs.FlashingReader_Read_Data_128Byte_1[10];
	PlcInputs.FlashingReader_Read_Data_128Byte_1[11] := HwInputs.FlashingReader_Read_Data_128Byte_1[11];
	PlcInputs.FlashingReader_Read_Data_128Byte_1[12] := HwInputs.FlashingReader_Read_Data_128Byte_1[12];
	PlcInputs.FlashingReader_Read_Data_128Byte_1[13] := HwInputs.FlashingReader_Read_Data_128Byte_1[13];
	PlcInputs.FlashingReader_Read_Data_128Byte_1[14] := HwInputs.FlashingReader_Read_Data_128Byte_1[14];
	PlcInputs.FlashingReader_Read_Data_128Byte_1[15] := HwInputs.FlashingReader_Read_Data_128Byte_1[15];
	PlcInputs.FlashingReader_Read_Data_128Byte_1[16] := HwInputs.FlashingReader_Read_Data_128Byte_1[16];
	PlcInputs.FlashingReader_Read_Data_128Byte_1[17] := HwInputs.FlashingReader_Read_Data_128Byte_1[17];
	PlcInputs.FlashingReader_Read_Data_128Byte_1[18] := HwInputs.FlashingReader_Read_Data_128Byte_1[18];
	PlcInputs.FlashingReader_Read_Data_128Byte_1[19] := HwInputs.FlashingReader_Read_Data_128Byte_1[19];
	PlcInputs.FlashingReader_Read_Data_128Byte_1[20] := HwInputs.FlashingReader_Read_Data_128Byte_1[20];
	PlcInputs.FlashingReader_Read_Data_128Byte_1[21] := HwInputs.FlashingReader_Read_Data_128Byte_1[21];
	PlcInputs.FlashingReader_Read_Data_128Byte_1[22] := HwInputs.FlashingReader_Read_Data_128Byte_1[22];
	PlcInputs.FlashingReader_Read_Data_128Byte_1[23] := HwInputs.FlashingReader_Read_Data_128Byte_1[23];
	PlcInputs.FlashingReader_Read_Data_128Byte_1[24] := HwInputs.FlashingReader_Read_Data_128Byte_1[24];
	PlcInputs.FlashingReader_Read_Data_128Byte_1[25] := HwInputs.FlashingReader_Read_Data_128Byte_1[25];
	PlcInputs.FlashingReader_Read_Data_128Byte_1[26] := HwInputs.FlashingReader_Read_Data_128Byte_1[26];
	PlcInputs.FlashingReader_Read_Data_128Byte_1[27] := HwInputs.FlashingReader_Read_Data_128Byte_1[27];
	PlcInputs.FlashingReader_Read_Data_128Byte_1[28] := HwInputs.FlashingReader_Read_Data_128Byte_1[28];
	PlcInputs.FlashingReader_Read_Data_128Byte_1[29] := HwInputs.FlashingReader_Read_Data_128Byte_1[29];
	PlcInputs.FlashingReader_Read_Data_128Byte_1[30] := HwInputs.FlashingReader_Read_Data_128Byte_1[30];
	PlcInputs.FlashingReader_Read_Data_128Byte_1[31] := HwInputs.FlashingReader_Read_Data_128Byte_1[31];
	PlcInputs.FlashingReader_Read_Data_128Byte_1[32] := HwInputs.FlashingReader_Read_Data_128Byte_1[32];
	PlcInputs.FlashingReader_Read_Data_128Byte_1[33] := HwInputs.FlashingReader_Read_Data_128Byte_1[33];
	PlcInputs.FlashingReader_Read_Data_128Byte_1[34] := HwInputs.FlashingReader_Read_Data_128Byte_1[34];
	PlcInputs.FlashingReader_Read_Data_128Byte_1[35] := HwInputs.FlashingReader_Read_Data_128Byte_1[35];
	PlcInputs.FlashingReader_Read_Data_128Byte_1[36] := HwInputs.FlashingReader_Read_Data_128Byte_1[36];
	PlcInputs.FlashingReader_Read_Data_128Byte_1[37] := HwInputs.FlashingReader_Read_Data_128Byte_1[37];
	PlcInputs.FlashingReader_Read_Data_128Byte_1[38] := HwInputs.FlashingReader_Read_Data_128Byte_1[38];
	PlcInputs.FlashingReader_Read_Data_128Byte_1[39] := HwInputs.FlashingReader_Read_Data_128Byte_1[39];
	PlcInputs.FlashingReader_Read_Data_128Byte_1[40] := HwInputs.FlashingReader_Read_Data_128Byte_1[40];
	PlcInputs.FlashingReader_Read_Data_128Byte_1[41] := HwInputs.FlashingReader_Read_Data_128Byte_1[41];
	PlcInputs.FlashingReader_Read_Data_128Byte_1[42] := HwInputs.FlashingReader_Read_Data_128Byte_1[42];
	PlcInputs.FlashingReader_Read_Data_128Byte_1[43] := HwInputs.FlashingReader_Read_Data_128Byte_1[43];
	PlcInputs.FlashingReader_Read_Data_128Byte_1[44] := HwInputs.FlashingReader_Read_Data_128Byte_1[44];
	PlcInputs.FlashingReader_Read_Data_128Byte_1[45] := HwInputs.FlashingReader_Read_Data_128Byte_1[45];
	PlcInputs.FlashingReader_Read_Data_128Byte_1[46] := HwInputs.FlashingReader_Read_Data_128Byte_1[46];
	PlcInputs.FlashingReader_Read_Data_128Byte_1[47] := HwInputs.FlashingReader_Read_Data_128Byte_1[47];
	PlcInputs.FlashingReader_Read_Data_128Byte_1[48] := HwInputs.FlashingReader_Read_Data_128Byte_1[48];
	PlcInputs.FlashingReader_Read_Data_128Byte_1[49] := HwInputs.FlashingReader_Read_Data_128Byte_1[49];
	PlcInputs.FlashingReader_Read_Data_128Byte_1[50] := HwInputs.FlashingReader_Read_Data_128Byte_1[50];
	PlcInputs.FlashingReader_Read_Data_128Byte_1[51] := HwInputs.FlashingReader_Read_Data_128Byte_1[51];
	PlcInputs.FlashingReader_Read_Data_128Byte_1[52] := HwInputs.FlashingReader_Read_Data_128Byte_1[52];
	PlcInputs.FlashingReader_Read_Data_128Byte_1[53] := HwInputs.FlashingReader_Read_Data_128Byte_1[53];
	PlcInputs.FlashingReader_Read_Data_128Byte_1[54] := HwInputs.FlashingReader_Read_Data_128Byte_1[54];
	PlcInputs.FlashingReader_Read_Data_128Byte_1[55] := HwInputs.FlashingReader_Read_Data_128Byte_1[55];
	PlcInputs.FlashingReader_Read_Data_128Byte_1[56] := HwInputs.FlashingReader_Read_Data_128Byte_1[56];
	PlcInputs.FlashingReader_Read_Data_128Byte_1[57] := HwInputs.FlashingReader_Read_Data_128Byte_1[57];
	PlcInputs.FlashingReader_Read_Data_128Byte_1[58] := HwInputs.FlashingReader_Read_Data_128Byte_1[58];
	PlcInputs.FlashingReader_Read_Data_128Byte_1[59] := HwInputs.FlashingReader_Read_Data_128Byte_1[59];
	PlcInputs.FlashingReader_Read_Data_128Byte_1[60] := HwInputs.FlashingReader_Read_Data_128Byte_1[60];
	PlcInputs.FlashingReader_Read_Data_128Byte_1[61] := HwInputs.FlashingReader_Read_Data_128Byte_1[61];
	PlcInputs.FlashingReader_Read_Data_128Byte_1[62] := HwInputs.FlashingReader_Read_Data_128Byte_1[62];
	PlcInputs.FlashingReader_Read_Data_128Byte_1[63] := HwInputs.FlashingReader_Read_Data_128Byte_1[63];
	PlcInputs.FlashingReader_Read_Data_128Byte_1[64] := HwInputs.FlashingReader_Read_Data_128Byte_1[64];
	PlcInputs.FlashingReader_Read_Data_128Byte_1[65] := HwInputs.FlashingReader_Read_Data_128Byte_1[65];
	PlcInputs.FlashingReader_Read_Data_128Byte_1[66] := HwInputs.FlashingReader_Read_Data_128Byte_1[66];
	PlcInputs.FlashingReader_Read_Data_128Byte_1[67] := HwInputs.FlashingReader_Read_Data_128Byte_1[67];
	PlcInputs.FlashingReader_Read_Data_128Byte_1[68] := HwInputs.FlashingReader_Read_Data_128Byte_1[68];
	PlcInputs.FlashingReader_Read_Data_128Byte_1[69] := HwInputs.FlashingReader_Read_Data_128Byte_1[69];
	PlcInputs.FlashingReader_Read_Data_128Byte_1[70] := HwInputs.FlashingReader_Read_Data_128Byte_1[70];
	PlcInputs.FlashingReader_Read_Data_128Byte_1[71] := HwInputs.FlashingReader_Read_Data_128Byte_1[71];
	PlcInputs.FlashingReader_Read_Data_128Byte_1[72] := HwInputs.FlashingReader_Read_Data_128Byte_1[72];
	PlcInputs.FlashingReader_Read_Data_128Byte_1[73] := HwInputs.FlashingReader_Read_Data_128Byte_1[73];
	PlcInputs.FlashingReader_Read_Data_128Byte_1[74] := HwInputs.FlashingReader_Read_Data_128Byte_1[74];
	PlcInputs.FlashingReader_Read_Data_128Byte_1[75] := HwInputs.FlashingReader_Read_Data_128Byte_1[75];
	PlcInputs.FlashingReader_Read_Data_128Byte_1[76] := HwInputs.FlashingReader_Read_Data_128Byte_1[76];
	PlcInputs.FlashingReader_Read_Data_128Byte_1[77] := HwInputs.FlashingReader_Read_Data_128Byte_1[77];
	PlcInputs.FlashingReader_Read_Data_128Byte_1[78] := HwInputs.FlashingReader_Read_Data_128Byte_1[78];
	PlcInputs.FlashingReader_Read_Data_128Byte_1[79] := HwInputs.FlashingReader_Read_Data_128Byte_1[79];
	PlcInputs.FlashingReader_Read_Data_128Byte_1[80] := HwInputs.FlashingReader_Read_Data_128Byte_1[80];
	PlcInputs.FlashingReader_Read_Data_128Byte_1[81] := HwInputs.FlashingReader_Read_Data_128Byte_1[81];
	PlcInputs.FlashingReader_Read_Data_128Byte_1[82] := HwInputs.FlashingReader_Read_Data_128Byte_1[82];
	PlcInputs.FlashingReader_Read_Data_128Byte_1[83] := HwInputs.FlashingReader_Read_Data_128Byte_1[83];
	PlcInputs.FlashingReader_Read_Data_128Byte_1[84] := HwInputs.FlashingReader_Read_Data_128Byte_1[84];
	PlcInputs.FlashingReader_Read_Data_128Byte_1[85] := HwInputs.FlashingReader_Read_Data_128Byte_1[85];
	PlcInputs.FlashingReader_Read_Data_128Byte_1[86] := HwInputs.FlashingReader_Read_Data_128Byte_1[86];
	PlcInputs.FlashingReader_Read_Data_128Byte_1[87] := HwInputs.FlashingReader_Read_Data_128Byte_1[87];
	PlcInputs.FlashingReader_Read_Data_128Byte_1[88] := HwInputs.FlashingReader_Read_Data_128Byte_1[88];
	PlcInputs.FlashingReader_Read_Data_128Byte_1[89] := HwInputs.FlashingReader_Read_Data_128Byte_1[89];
	PlcInputs.FlashingReader_Read_Data_128Byte_1[90] := HwInputs.FlashingReader_Read_Data_128Byte_1[90];
	PlcInputs.FlashingReader_Read_Data_128Byte_1[91] := HwInputs.FlashingReader_Read_Data_128Byte_1[91];
	PlcInputs.FlashingReader_Read_Data_128Byte_1[92] := HwInputs.FlashingReader_Read_Data_128Byte_1[92];
	PlcInputs.FlashingReader_Read_Data_128Byte_1[93] := HwInputs.FlashingReader_Read_Data_128Byte_1[93];
	PlcInputs.FlashingReader_Read_Data_128Byte_1[94] := HwInputs.FlashingReader_Read_Data_128Byte_1[94];
	PlcInputs.FlashingReader_Read_Data_128Byte_1[95] := HwInputs.FlashingReader_Read_Data_128Byte_1[95];
	PlcInputs.FlashingReader_Read_Data_128Byte_1[96] := HwInputs.FlashingReader_Read_Data_128Byte_1[96];
	PlcInputs.FlashingReader_Read_Data_128Byte_1[97] := HwInputs.FlashingReader_Read_Data_128Byte_1[97];
	PlcInputs.FlashingReader_Read_Data_128Byte_1[98] := HwInputs.FlashingReader_Read_Data_128Byte_1[98];
	PlcInputs.FlashingReader_Read_Data_128Byte_1[99] := HwInputs.FlashingReader_Read_Data_128Byte_1[99];
	PlcInputs.FlashingReader_Read_Data_128Byte_1[100] := HwInputs.FlashingReader_Read_Data_128Byte_1[100];
	PlcInputs.FlashingReader_Read_Data_128Byte_1[101] := HwInputs.FlashingReader_Read_Data_128Byte_1[101];
	PlcInputs.FlashingReader_Read_Data_128Byte_1[102] := HwInputs.FlashingReader_Read_Data_128Byte_1[102];
	PlcInputs.FlashingReader_Read_Data_128Byte_1[103] := HwInputs.FlashingReader_Read_Data_128Byte_1[103];
	PlcInputs.FlashingReader_Read_Data_128Byte_1[104] := HwInputs.FlashingReader_Read_Data_128Byte_1[104];
	PlcInputs.FlashingReader_Read_Data_128Byte_1[105] := HwInputs.FlashingReader_Read_Data_128Byte_1[105];
	PlcInputs.FlashingReader_Read_Data_128Byte_1[106] := HwInputs.FlashingReader_Read_Data_128Byte_1[106];
	PlcInputs.FlashingReader_Read_Data_128Byte_1[107] := HwInputs.FlashingReader_Read_Data_128Byte_1[107];
	PlcInputs.FlashingReader_Read_Data_128Byte_1[108] := HwInputs.FlashingReader_Read_Data_128Byte_1[108];
	PlcInputs.FlashingReader_Read_Data_128Byte_1[109] := HwInputs.FlashingReader_Read_Data_128Byte_1[109];
	PlcInputs.FlashingReader_Read_Data_128Byte_1[110] := HwInputs.FlashingReader_Read_Data_128Byte_1[110];
	PlcInputs.FlashingReader_Read_Data_128Byte_1[111] := HwInputs.FlashingReader_Read_Data_128Byte_1[111];
	PlcInputs.FlashingReader_Read_Data_128Byte_1[112] := HwInputs.FlashingReader_Read_Data_128Byte_1[112];
	PlcInputs.FlashingReader_Read_Data_128Byte_1[113] := HwInputs.FlashingReader_Read_Data_128Byte_1[113];
	PlcInputs.FlashingReader_Read_Data_128Byte_1[114] := HwInputs.FlashingReader_Read_Data_128Byte_1[114];
	PlcInputs.FlashingReader_Read_Data_128Byte_1[115] := HwInputs.FlashingReader_Read_Data_128Byte_1[115];
	PlcInputs.FlashingReader_Read_Data_128Byte_1[116] := HwInputs.FlashingReader_Read_Data_128Byte_1[116];
	PlcInputs.FlashingReader_Read_Data_128Byte_1[117] := HwInputs.FlashingReader_Read_Data_128Byte_1[117];
	PlcInputs.FlashingReader_Read_Data_128Byte_1[118] := HwInputs.FlashingReader_Read_Data_128Byte_1[118];
	PlcInputs.FlashingReader_Read_Data_128Byte_1[119] := HwInputs.FlashingReader_Read_Data_128Byte_1[119];
	PlcInputs.FlashingReader_Read_Data_128Byte_1[120] := HwInputs.FlashingReader_Read_Data_128Byte_1[120];
	PlcInputs.FlashingReader_Read_Data_128Byte_1[121] := HwInputs.FlashingReader_Read_Data_128Byte_1[121];
	PlcInputs.FlashingReader_Read_Data_128Byte_1[122] := HwInputs.FlashingReader_Read_Data_128Byte_1[122];
	PlcInputs.FlashingReader_Read_Data_128Byte_1[123] := HwInputs.FlashingReader_Read_Data_128Byte_1[123];
	PlcInputs.FlashingReader_Read_Data_128Byte_1[124] := HwInputs.FlashingReader_Read_Data_128Byte_1[124];
	PlcInputs.FlashingReader_Read_Data_128Byte_1[125] := HwInputs.FlashingReader_Read_Data_128Byte_1[125];
	PlcInputs.FlashingReader_Read_Data_128Byte_1[126] := HwInputs.FlashingReader_Read_Data_128Byte_1[126];
	PlcInputs.FlashingReader_Read_Data_128Byte_1[127] := HwInputs.FlashingReader_Read_Data_128Byte_1[127];
	PlcInputs.FlashingReader_Read_Data_128Byte_1[128] := HwInputs.FlashingReader_Read_Data_128Byte_1[128];
	PlcInputs.FlashingReader_Read_Data_128Byte_1[129] := HwInputs.FlashingReader_Read_Data_128Byte_1[129];
	PlcInputs.FlashingReader_Read_Data_128Byte_1[130] := HwInputs.FlashingReader_Read_Data_128Byte_1[130];
	PlcInputs.FlashingReader_Read_Data_128Byte_1[131] := HwInputs.FlashingReader_Read_Data_128Byte_1[131];
	PlcInputs.FlashingReader_Read_Data_128Byte_1[132] := HwInputs.FlashingReader_Read_Data_128Byte_1[132];
	PlcInputs.FlashingReader_Read_Data_128Byte_1[133] := HwInputs.FlashingReader_Read_Data_128Byte_1[133];
	PlcInputs.FlashingReader_Read_Data_128Byte_1[134] := HwInputs.FlashingReader_Read_Data_128Byte_1[134];
	PlcInputs.FlashingReader_Read_Data_128Byte_1[135] := HwInputs.FlashingReader_Read_Data_128Byte_1[135];
	PlcInputs.AS10_2flashing_In_64_Byte_1[0] := HwInputs.AS10_2flashing_In_64_Byte_1[0];
	PlcInputs.AS10_2flashing_In_64_Byte_1[1] := HwInputs.AS10_2flashing_In_64_Byte_1[1];
	PlcInputs.AS10_2flashing_In_64_Byte_1[2] := HwInputs.AS10_2flashing_In_64_Byte_1[2];
	PlcInputs.AS10_2flashing_In_64_Byte_1[3] := HwInputs.AS10_2flashing_In_64_Byte_1[3];
	PlcInputs.AS10_2flashing_In_64_Byte_1[4] := HwInputs.AS10_2flashing_In_64_Byte_1[4];
	PlcInputs.AS10_2flashing_In_64_Byte_1[5] := HwInputs.AS10_2flashing_In_64_Byte_1[5];
	PlcInputs.AS10_2flashing_In_64_Byte_1[6] := HwInputs.AS10_2flashing_In_64_Byte_1[6];
	PlcInputs.AS10_2flashing_In_64_Byte_1[7] := HwInputs.AS10_2flashing_In_64_Byte_1[7];
	PlcInputs.AS10_2flashing_In_64_Byte_1[8] := HwInputs.AS10_2flashing_In_64_Byte_1[8];
	PlcInputs.AS10_2flashing_In_64_Byte_1[9] := HwInputs.AS10_2flashing_In_64_Byte_1[9];
	PlcInputs.AS10_2flashing_In_64_Byte_1[10] := HwInputs.AS10_2flashing_In_64_Byte_1[10];
	PlcInputs.AS10_2flashing_In_64_Byte_1[11] := HwInputs.AS10_2flashing_In_64_Byte_1[11];
	PlcInputs.AS10_2flashing_In_64_Byte_1[12] := HwInputs.AS10_2flashing_In_64_Byte_1[12];
	PlcInputs.AS10_2flashing_In_64_Byte_1[13] := HwInputs.AS10_2flashing_In_64_Byte_1[13];
	PlcInputs.AS10_2flashing_In_64_Byte_1[14] := HwInputs.AS10_2flashing_In_64_Byte_1[14];
	PlcInputs.AS10_2flashing_In_64_Byte_1[15] := HwInputs.AS10_2flashing_In_64_Byte_1[15];
	PlcInputs.AS10_2flashing_In_64_Byte_1[16] := HwInputs.AS10_2flashing_In_64_Byte_1[16];
	PlcInputs.AS10_2flashing_In_64_Byte_1[17] := HwInputs.AS10_2flashing_In_64_Byte_1[17];
	PlcInputs.AS10_2flashing_In_64_Byte_1[18] := HwInputs.AS10_2flashing_In_64_Byte_1[18];
	PlcInputs.AS10_2flashing_In_64_Byte_1[19] := HwInputs.AS10_2flashing_In_64_Byte_1[19];
	PlcInputs.AS10_2flashing_In_64_Byte_1[20] := HwInputs.AS10_2flashing_In_64_Byte_1[20];
	PlcInputs.AS10_2flashing_In_64_Byte_1[21] := HwInputs.AS10_2flashing_In_64_Byte_1[21];
	PlcInputs.AS10_2flashing_In_64_Byte_1[22] := HwInputs.AS10_2flashing_In_64_Byte_1[22];
	PlcInputs.AS10_2flashing_In_64_Byte_1[23] := HwInputs.AS10_2flashing_In_64_Byte_1[23];
	PlcInputs.AS10_2flashing_In_64_Byte_1[24] := HwInputs.AS10_2flashing_In_64_Byte_1[24];
	PlcInputs.AS10_2flashing_In_64_Byte_1[25] := HwInputs.AS10_2flashing_In_64_Byte_1[25];
	PlcInputs.AS10_2flashing_In_64_Byte_1[26] := HwInputs.AS10_2flashing_In_64_Byte_1[26];
	PlcInputs.AS10_2flashing_In_64_Byte_1[27] := HwInputs.AS10_2flashing_In_64_Byte_1[27];
	PlcInputs.AS10_2flashing_In_64_Byte_1[28] := HwInputs.AS10_2flashing_In_64_Byte_1[28];
	PlcInputs.AS10_2flashing_In_64_Byte_1[29] := HwInputs.AS10_2flashing_In_64_Byte_1[29];
	PlcInputs.AS10_2flashing_In_64_Byte_1[30] := HwInputs.AS10_2flashing_In_64_Byte_1[30];
	PlcInputs.AS10_2flashing_In_64_Byte_1[31] := HwInputs.AS10_2flashing_In_64_Byte_1[31];
	PlcInputs.AS10_2flashing_In_64_Byte_1[32] := HwInputs.AS10_2flashing_In_64_Byte_1[32];
	PlcInputs.AS10_2flashing_In_64_Byte_1[33] := HwInputs.AS10_2flashing_In_64_Byte_1[33];
	PlcInputs.AS10_2flashing_In_64_Byte_1[34] := HwInputs.AS10_2flashing_In_64_Byte_1[34];
	PlcInputs.AS10_2flashing_In_64_Byte_1[35] := HwInputs.AS10_2flashing_In_64_Byte_1[35];
	PlcInputs.AS10_2flashing_In_64_Byte_1[36] := HwInputs.AS10_2flashing_In_64_Byte_1[36];
	PlcInputs.AS10_2flashing_In_64_Byte_1[37] := HwInputs.AS10_2flashing_In_64_Byte_1[37];
	PlcInputs.AS10_2flashing_In_64_Byte_1[38] := HwInputs.AS10_2flashing_In_64_Byte_1[38];
	PlcInputs.AS10_2flashing_In_64_Byte_1[39] := HwInputs.AS10_2flashing_In_64_Byte_1[39];
	PlcInputs.AS10_2flashing_In_64_Byte_1[40] := HwInputs.AS10_2flashing_In_64_Byte_1[40];
	PlcInputs.AS10_2flashing_In_64_Byte_1[41] := HwInputs.AS10_2flashing_In_64_Byte_1[41];
	PlcInputs.AS10_2flashing_In_64_Byte_1[42] := HwInputs.AS10_2flashing_In_64_Byte_1[42];
	PlcInputs.AS10_2flashing_In_64_Byte_1[43] := HwInputs.AS10_2flashing_In_64_Byte_1[43];
	PlcInputs.AS10_2flashing_In_64_Byte_1[44] := HwInputs.AS10_2flashing_In_64_Byte_1[44];
	PlcInputs.AS10_2flashing_In_64_Byte_1[45] := HwInputs.AS10_2flashing_In_64_Byte_1[45];
	PlcInputs.AS10_2flashing_In_64_Byte_1[46] := HwInputs.AS10_2flashing_In_64_Byte_1[46];
	PlcInputs.AS10_2flashing_In_64_Byte_1[47] := HwInputs.AS10_2flashing_In_64_Byte_1[47];
	PlcInputs.AS10_2flashing_In_64_Byte_1[48] := HwInputs.AS10_2flashing_In_64_Byte_1[48];
	PlcInputs.AS10_2flashing_In_64_Byte_1[49] := HwInputs.AS10_2flashing_In_64_Byte_1[49];
	PlcInputs.AS10_2flashing_In_64_Byte_1[50] := HwInputs.AS10_2flashing_In_64_Byte_1[50];
	PlcInputs.AS10_2flashing_In_64_Byte_1[51] := HwInputs.AS10_2flashing_In_64_Byte_1[51];
	PlcInputs.AS10_2flashing_In_64_Byte_1[52] := HwInputs.AS10_2flashing_In_64_Byte_1[52];
	PlcInputs.AS10_2flashing_In_64_Byte_1[53] := HwInputs.AS10_2flashing_In_64_Byte_1[53];
	PlcInputs.AS10_2flashing_In_64_Byte_1[54] := HwInputs.AS10_2flashing_In_64_Byte_1[54];
	PlcInputs.AS10_2flashing_In_64_Byte_1[55] := HwInputs.AS10_2flashing_In_64_Byte_1[55];
	PlcInputs.AS10_2flashing_In_64_Byte_1[56] := HwInputs.AS10_2flashing_In_64_Byte_1[56];
	PlcInputs.AS10_2flashing_In_64_Byte_1[57] := HwInputs.AS10_2flashing_In_64_Byte_1[57];
	PlcInputs.AS10_2flashing_In_64_Byte_1[58] := HwInputs.AS10_2flashing_In_64_Byte_1[58];
	PlcInputs.AS10_2flashing_In_64_Byte_1[59] := HwInputs.AS10_2flashing_In_64_Byte_1[59];
	PlcInputs.AS10_2flashing_In_64_Byte_1[60] := HwInputs.AS10_2flashing_In_64_Byte_1[60];
	PlcInputs.AS10_2flashing_In_64_Byte_1[61] := HwInputs.AS10_2flashing_In_64_Byte_1[61];
	PlcInputs.AS10_2flashing_In_64_Byte_1[62] := HwInputs.AS10_2flashing_In_64_Byte_1[62];
	PlcInputs.AS10_2flashing_In_64_Byte_1[63] := HwInputs.AS10_2flashing_In_64_Byte_1[63];
END_FUNCTION

(* ---- CopyOutputs.st ---- *)
FUNCTION CopyOutputs
	VAR_EXTERNAL
		HwOutputs : HwOutputs;
		PlcOutputs : PlcOutputs;
	END_VAR
	HwOutputs.CPX_PneuOst_AS11_MPA1S_VMPA1_FB_EMS_8_8DO_1 := PlcOutputs.CPX_PneuOst_AS11_MPA1S_VMPA1_FB_EMS_8_8DO_1;
	HwOutputs.CPX_PneuOst_AS11_MPA2S_VMPA2_FB_EMS_4_4DO_2 := PlcOutputs.CPX_PneuOst_AS11_MPA2S_VMPA2_FB_EMS_4_4DO_2;
	HwOutputs.CPX_PneuOst_AS11_MPA2S_VMPA2_FB_EMS_4_4DO_1 := PlcOutputs.CPX_PneuOst_AS11_MPA2S_VMPA2_FB_EMS_4_4DO_1;
	HwOutputs.CPX_PneuOst_AS11_MPA1S_VMPA1_FB_EMS_8_8DO_3 := PlcOutputs.CPX_PneuOst_AS11_MPA1S_VMPA1_FB_EMS_8_8DO_3;
	HwOutputs.CPX_PneuOst_AS11_MPA1S_VMPA1_FB_EMS_8_8DO_4 := PlcOutputs.CPX_PneuOst_AS11_MPA1S_VMPA1_FB_EMS_8_8DO_4;
	HwOutputs.CPX_PneuOst_AS11_MPA1G_VMPA1_FB_EMG_8_8DO_1 := PlcOutputs.CPX_PneuOst_AS11_MPA1G_VMPA1_FB_EMG_8_8DO_1;
	HwOutputs._6A2_AS11_6A5 := PlcOutputs._6A2_AS11_6A5;
	HwOutputs._6A2_AS11_6A13[0] := PlcOutputs._6A2_AS11_6A13[0];
	HwOutputs._6A2_AS11_6A13[1] := PlcOutputs._6A2_AS11_6A13[1];
	HwOutputs._6A2_AS11_6A13[2] := PlcOutputs._6A2_AS11_6A13[2];
	HwOutputs._6A2_AS11_6A13[3] := PlcOutputs._6A2_AS11_6A13[3];
	HwOutputs._6A2_AS11_6A13[4] := PlcOutputs._6A2_AS11_6A13[4];
	HwOutputs._6A2_AS11_6A13[5] := PlcOutputs._6A2_AS11_6A13[5];
	HwOutputs._6A2_AS11_6A13[6] := PlcOutputs._6A2_AS11_6A13[6];
	HwOutputs._6A2_AS11_6A13[7] := PlcOutputs._6A2_AS11_6A13[7];
	HwOutputs._6A2_AS11_6A13[8] := PlcOutputs._6A2_AS11_6A13[8];
	HwOutputs._6A2_AS11_6A13[9] := PlcOutputs._6A2_AS11_6A13[9];
	HwOutputs._6A2_AS11_6A13[10] := PlcOutputs._6A2_AS11_6A13[10];
	HwOutputs._6A2_AS11_6A13[11] := PlcOutputs._6A2_AS11_6A13[11];
	HwOutputs._6A2_AS11_6A13[12] := PlcOutputs._6A2_AS11_6A13[12];
	HwOutputs._6A2_AS11_6A13[13] := PlcOutputs._6A2_AS11_6A13[13];
	HwOutputs._6A2_AS11_6A13[14] := PlcOutputs._6A2_AS11_6A13[14];
	HwOutputs._6A2_AS11_6A13[15] := PlcOutputs._6A2_AS11_6A13[15];
	HwOutputs._6A2_AS11_6A13[16] := PlcOutputs._6A2_AS11_6A13[16];
	HwOutputs._6A2_AS11_6A13[17] := PlcOutputs._6A2_AS11_6A13[17];
	HwOutputs._6A2_AS11_6A13[18] := PlcOutputs._6A2_AS11_6A13[18];
	HwOutputs._6A2_AS11_6A13[19] := PlcOutputs._6A2_AS11_6A13[19];
	HwOutputs._6A2_AS11_6A13[20] := PlcOutputs._6A2_AS11_6A13[20];
	HwOutputs._6A2_AS11_6A13[21] := PlcOutputs._6A2_AS11_6A13[21];
	HwOutputs._6A2_AS11_6A13[22] := PlcOutputs._6A2_AS11_6A13[22];
	HwOutputs._6A2_AS11_6A13[23] := PlcOutputs._6A2_AS11_6A13[23];
	HwOutputs._6A2_AS11_6A13[24] := PlcOutputs._6A2_AS11_6A13[24];
	HwOutputs._6A2_AS11_6A13[25] := PlcOutputs._6A2_AS11_6A13[25];
	HwOutputs._6A2_AS11_6A13[26] := PlcOutputs._6A2_AS11_6A13[26];
	HwOutputs._6A2_AS11_6A13[27] := PlcOutputs._6A2_AS11_6A13[27];
	HwOutputs._6A2_AS11_6A13[28] := PlcOutputs._6A2_AS11_6A13[28];
	HwOutputs._6A2_AS11_6A13[29] := PlcOutputs._6A2_AS11_6A13[29];
	HwOutputs._6A2_AS11_6A13[30] := PlcOutputs._6A2_AS11_6A13[30];
	HwOutputs._6A2_AS11_6A13[31] := PlcOutputs._6A2_AS11_6A13[31];
	HwOutputs._6A2_AS11_6A20[0] := PlcOutputs._6A2_AS11_6A20[0];
	HwOutputs._6A2_AS11_6A20[1] := PlcOutputs._6A2_AS11_6A20[1];
	HwOutputs._6A2_AS11_6A20[2] := PlcOutputs._6A2_AS11_6A20[2];
	HwOutputs._6A2_AS11_6A20[3] := PlcOutputs._6A2_AS11_6A20[3];
	HwOutputs._6A2_AS11_6A20[4] := PlcOutputs._6A2_AS11_6A20[4];
	HwOutputs._6A2_AS11_6A20[5] := PlcOutputs._6A2_AS11_6A20[5];
	HwOutputs._6A2_AS11_6A20[6] := PlcOutputs._6A2_AS11_6A20[6];
	HwOutputs._6A2_AS11_6A20[7] := PlcOutputs._6A2_AS11_6A20[7];
	HwOutputs.HousingReader_AS11_Latch_and_Error_Clear_Control_Bits_1 := PlcOutputs.HousingReader_AS11_Latch_and_Error_Clear_Control_Bits_1;
	HwOutputs.HousingReader_AS11_Operation_instruction_Control_Bits_1 := PlcOutputs.HousingReader_AS11_Operation_instruction_Control_Bits_1;
	HwOutputs.HousingReader_AS11_Completion_Clear_Control_Bits_1 := PlcOutputs.HousingReader_AS11_Completion_Clear_Control_Bits_1;
	HwOutputs.HousingReader_AS11_Parameter_Bank_Number_1 := PlcOutputs.HousingReader_AS11_Parameter_Bank_Number_1;
	HwOutputs.HousingReader_AS11_User_Data_128Byte_1[0] := PlcOutputs.HousingReader_AS11_User_Data_128Byte_1[0];
	HwOutputs.HousingReader_AS11_User_Data_128Byte_1[1] := PlcOutputs.HousingReader_AS11_User_Data_128Byte_1[1];
	HwOutputs.HousingReader_AS11_User_Data_128Byte_1[2] := PlcOutputs.HousingReader_AS11_User_Data_128Byte_1[2];
	HwOutputs.HousingReader_AS11_User_Data_128Byte_1[3] := PlcOutputs.HousingReader_AS11_User_Data_128Byte_1[3];
	HwOutputs.HousingReader_AS11_User_Data_128Byte_1[4] := PlcOutputs.HousingReader_AS11_User_Data_128Byte_1[4];
	HwOutputs.HousingReader_AS11_User_Data_128Byte_1[5] := PlcOutputs.HousingReader_AS11_User_Data_128Byte_1[5];
	HwOutputs.HousingReader_AS11_User_Data_128Byte_1[6] := PlcOutputs.HousingReader_AS11_User_Data_128Byte_1[6];
	HwOutputs.HousingReader_AS11_User_Data_128Byte_1[7] := PlcOutputs.HousingReader_AS11_User_Data_128Byte_1[7];
	HwOutputs.HousingReader_AS11_User_Data_128Byte_1[8] := PlcOutputs.HousingReader_AS11_User_Data_128Byte_1[8];
	HwOutputs.HousingReader_AS11_User_Data_128Byte_1[9] := PlcOutputs.HousingReader_AS11_User_Data_128Byte_1[9];
	HwOutputs.HousingReader_AS11_User_Data_128Byte_1[10] := PlcOutputs.HousingReader_AS11_User_Data_128Byte_1[10];
	HwOutputs.HousingReader_AS11_User_Data_128Byte_1[11] := PlcOutputs.HousingReader_AS11_User_Data_128Byte_1[11];
	HwOutputs.HousingReader_AS11_User_Data_128Byte_1[12] := PlcOutputs.HousingReader_AS11_User_Data_128Byte_1[12];
	HwOutputs.HousingReader_AS11_User_Data_128Byte_1[13] := PlcOutputs.HousingReader_AS11_User_Data_128Byte_1[13];
	HwOutputs.HousingReader_AS11_User_Data_128Byte_1[14] := PlcOutputs.HousingReader_AS11_User_Data_128Byte_1[14];
	HwOutputs.HousingReader_AS11_User_Data_128Byte_1[15] := PlcOutputs.HousingReader_AS11_User_Data_128Byte_1[15];
	HwOutputs.HousingReader_AS11_User_Data_128Byte_1[16] := PlcOutputs.HousingReader_AS11_User_Data_128Byte_1[16];
	HwOutputs.HousingReader_AS11_User_Data_128Byte_1[17] := PlcOutputs.HousingReader_AS11_User_Data_128Byte_1[17];
	HwOutputs.HousingReader_AS11_User_Data_128Byte_1[18] := PlcOutputs.HousingReader_AS11_User_Data_128Byte_1[18];
	HwOutputs.HousingReader_AS11_User_Data_128Byte_1[19] := PlcOutputs.HousingReader_AS11_User_Data_128Byte_1[19];
	HwOutputs.HousingReader_AS11_User_Data_128Byte_1[20] := PlcOutputs.HousingReader_AS11_User_Data_128Byte_1[20];
	HwOutputs.HousingReader_AS11_User_Data_128Byte_1[21] := PlcOutputs.HousingReader_AS11_User_Data_128Byte_1[21];
	HwOutputs.HousingReader_AS11_User_Data_128Byte_1[22] := PlcOutputs.HousingReader_AS11_User_Data_128Byte_1[22];
	HwOutputs.HousingReader_AS11_User_Data_128Byte_1[23] := PlcOutputs.HousingReader_AS11_User_Data_128Byte_1[23];
	HwOutputs.HousingReader_AS11_User_Data_128Byte_1[24] := PlcOutputs.HousingReader_AS11_User_Data_128Byte_1[24];
	HwOutputs.HousingReader_AS11_User_Data_128Byte_1[25] := PlcOutputs.HousingReader_AS11_User_Data_128Byte_1[25];
	HwOutputs.HousingReader_AS11_User_Data_128Byte_1[26] := PlcOutputs.HousingReader_AS11_User_Data_128Byte_1[26];
	HwOutputs.HousingReader_AS11_User_Data_128Byte_1[27] := PlcOutputs.HousingReader_AS11_User_Data_128Byte_1[27];
	HwOutputs.HousingReader_AS11_User_Data_128Byte_1[28] := PlcOutputs.HousingReader_AS11_User_Data_128Byte_1[28];
	HwOutputs.HousingReader_AS11_User_Data_128Byte_1[29] := PlcOutputs.HousingReader_AS11_User_Data_128Byte_1[29];
	HwOutputs.HousingReader_AS11_User_Data_128Byte_1[30] := PlcOutputs.HousingReader_AS11_User_Data_128Byte_1[30];
	HwOutputs.HousingReader_AS11_User_Data_128Byte_1[31] := PlcOutputs.HousingReader_AS11_User_Data_128Byte_1[31];
	HwOutputs.HousingReader_AS11_User_Data_128Byte_1[32] := PlcOutputs.HousingReader_AS11_User_Data_128Byte_1[32];
	HwOutputs.HousingReader_AS11_User_Data_128Byte_1[33] := PlcOutputs.HousingReader_AS11_User_Data_128Byte_1[33];
	HwOutputs.HousingReader_AS11_User_Data_128Byte_1[34] := PlcOutputs.HousingReader_AS11_User_Data_128Byte_1[34];
	HwOutputs.HousingReader_AS11_User_Data_128Byte_1[35] := PlcOutputs.HousingReader_AS11_User_Data_128Byte_1[35];
	HwOutputs.HousingReader_AS11_User_Data_128Byte_1[36] := PlcOutputs.HousingReader_AS11_User_Data_128Byte_1[36];
	HwOutputs.HousingReader_AS11_User_Data_128Byte_1[37] := PlcOutputs.HousingReader_AS11_User_Data_128Byte_1[37];
	HwOutputs.HousingReader_AS11_User_Data_128Byte_1[38] := PlcOutputs.HousingReader_AS11_User_Data_128Byte_1[38];
	HwOutputs.HousingReader_AS11_User_Data_128Byte_1[39] := PlcOutputs.HousingReader_AS11_User_Data_128Byte_1[39];
	HwOutputs.HousingReader_AS11_User_Data_128Byte_1[40] := PlcOutputs.HousingReader_AS11_User_Data_128Byte_1[40];
	HwOutputs.HousingReader_AS11_User_Data_128Byte_1[41] := PlcOutputs.HousingReader_AS11_User_Data_128Byte_1[41];
	HwOutputs.HousingReader_AS11_User_Data_128Byte_1[42] := PlcOutputs.HousingReader_AS11_User_Data_128Byte_1[42];
	HwOutputs.HousingReader_AS11_User_Data_128Byte_1[43] := PlcOutputs.HousingReader_AS11_User_Data_128Byte_1[43];
	HwOutputs.HousingReader_AS11_User_Data_128Byte_1[44] := PlcOutputs.HousingReader_AS11_User_Data_128Byte_1[44];
	HwOutputs.HousingReader_AS11_User_Data_128Byte_1[45] := PlcOutputs.HousingReader_AS11_User_Data_128Byte_1[45];
	HwOutputs.HousingReader_AS11_User_Data_128Byte_1[46] := PlcOutputs.HousingReader_AS11_User_Data_128Byte_1[46];
	HwOutputs.HousingReader_AS11_User_Data_128Byte_1[47] := PlcOutputs.HousingReader_AS11_User_Data_128Byte_1[47];
	HwOutputs.HousingReader_AS11_User_Data_128Byte_1[48] := PlcOutputs.HousingReader_AS11_User_Data_128Byte_1[48];
	HwOutputs.HousingReader_AS11_User_Data_128Byte_1[49] := PlcOutputs.HousingReader_AS11_User_Data_128Byte_1[49];
	HwOutputs.HousingReader_AS11_User_Data_128Byte_1[50] := PlcOutputs.HousingReader_AS11_User_Data_128Byte_1[50];
	HwOutputs.HousingReader_AS11_User_Data_128Byte_1[51] := PlcOutputs.HousingReader_AS11_User_Data_128Byte_1[51];
	HwOutputs.HousingReader_AS11_User_Data_128Byte_1[52] := PlcOutputs.HousingReader_AS11_User_Data_128Byte_1[52];
	HwOutputs.HousingReader_AS11_User_Data_128Byte_1[53] := PlcOutputs.HousingReader_AS11_User_Data_128Byte_1[53];
	HwOutputs.HousingReader_AS11_User_Data_128Byte_1[54] := PlcOutputs.HousingReader_AS11_User_Data_128Byte_1[54];
	HwOutputs.HousingReader_AS11_User_Data_128Byte_1[55] := PlcOutputs.HousingReader_AS11_User_Data_128Byte_1[55];
	HwOutputs.HousingReader_AS11_User_Data_128Byte_1[56] := PlcOutputs.HousingReader_AS11_User_Data_128Byte_1[56];
	HwOutputs.HousingReader_AS11_User_Data_128Byte_1[57] := PlcOutputs.HousingReader_AS11_User_Data_128Byte_1[57];
	HwOutputs.HousingReader_AS11_User_Data_128Byte_1[58] := PlcOutputs.HousingReader_AS11_User_Data_128Byte_1[58];
	HwOutputs.HousingReader_AS11_User_Data_128Byte_1[59] := PlcOutputs.HousingReader_AS11_User_Data_128Byte_1[59];
	HwOutputs.HousingReader_AS11_User_Data_128Byte_1[60] := PlcOutputs.HousingReader_AS11_User_Data_128Byte_1[60];
	HwOutputs.HousingReader_AS11_User_Data_128Byte_1[61] := PlcOutputs.HousingReader_AS11_User_Data_128Byte_1[61];
	HwOutputs.HousingReader_AS11_User_Data_128Byte_1[62] := PlcOutputs.HousingReader_AS11_User_Data_128Byte_1[62];
	HwOutputs.HousingReader_AS11_User_Data_128Byte_1[63] := PlcOutputs.HousingReader_AS11_User_Data_128Byte_1[63];
	HwOutputs.HousingReader_AS11_User_Data_128Byte_1[64] := PlcOutputs.HousingReader_AS11_User_Data_128Byte_1[64];
	HwOutputs.HousingReader_AS11_User_Data_128Byte_1[65] := PlcOutputs.HousingReader_AS11_User_Data_128Byte_1[65];
	HwOutputs.HousingReader_AS11_User_Data_128Byte_1[66] := PlcOutputs.HousingReader_AS11_User_Data_128Byte_1[66];
	HwOutputs.HousingReader_AS11_User_Data_128Byte_1[67] := PlcOutputs.HousingReader_AS11_User_Data_128Byte_1[67];
	HwOutputs.HousingReader_AS11_User_Data_128Byte_1[68] := PlcOutputs.HousingReader_AS11_User_Data_128Byte_1[68];
	HwOutputs.HousingReader_AS11_User_Data_128Byte_1[69] := PlcOutputs.HousingReader_AS11_User_Data_128Byte_1[69];
	HwOutputs.HousingReader_AS11_User_Data_128Byte_1[70] := PlcOutputs.HousingReader_AS11_User_Data_128Byte_1[70];
	HwOutputs.HousingReader_AS11_User_Data_128Byte_1[71] := PlcOutputs.HousingReader_AS11_User_Data_128Byte_1[71];
	HwOutputs.HousingReader_AS11_User_Data_128Byte_1[72] := PlcOutputs.HousingReader_AS11_User_Data_128Byte_1[72];
	HwOutputs.HousingReader_AS11_User_Data_128Byte_1[73] := PlcOutputs.HousingReader_AS11_User_Data_128Byte_1[73];
	HwOutputs.HousingReader_AS11_User_Data_128Byte_1[74] := PlcOutputs.HousingReader_AS11_User_Data_128Byte_1[74];
	HwOutputs.HousingReader_AS11_User_Data_128Byte_1[75] := PlcOutputs.HousingReader_AS11_User_Data_128Byte_1[75];
	HwOutputs.HousingReader_AS11_User_Data_128Byte_1[76] := PlcOutputs.HousingReader_AS11_User_Data_128Byte_1[76];
	HwOutputs.HousingReader_AS11_User_Data_128Byte_1[77] := PlcOutputs.HousingReader_AS11_User_Data_128Byte_1[77];
	HwOutputs.HousingReader_AS11_User_Data_128Byte_1[78] := PlcOutputs.HousingReader_AS11_User_Data_128Byte_1[78];
	HwOutputs.HousingReader_AS11_User_Data_128Byte_1[79] := PlcOutputs.HousingReader_AS11_User_Data_128Byte_1[79];
	HwOutputs.HousingReader_AS11_User_Data_128Byte_1[80] := PlcOutputs.HousingReader_AS11_User_Data_128Byte_1[80];
	HwOutputs.HousingReader_AS11_User_Data_128Byte_1[81] := PlcOutputs.HousingReader_AS11_User_Data_128Byte_1[81];
	HwOutputs.HousingReader_AS11_User_Data_128Byte_1[82] := PlcOutputs.HousingReader_AS11_User_Data_128Byte_1[82];
	HwOutputs.HousingReader_AS11_User_Data_128Byte_1[83] := PlcOutputs.HousingReader_AS11_User_Data_128Byte_1[83];
	HwOutputs.HousingReader_AS11_User_Data_128Byte_1[84] := PlcOutputs.HousingReader_AS11_User_Data_128Byte_1[84];
	HwOutputs.HousingReader_AS11_User_Data_128Byte_1[85] := PlcOutputs.HousingReader_AS11_User_Data_128Byte_1[85];
	HwOutputs.HousingReader_AS11_User_Data_128Byte_1[86] := PlcOutputs.HousingReader_AS11_User_Data_128Byte_1[86];
	HwOutputs.HousingReader_AS11_User_Data_128Byte_1[87] := PlcOutputs.HousingReader_AS11_User_Data_128Byte_1[87];
	HwOutputs.HousingReader_AS11_User_Data_128Byte_1[88] := PlcOutputs.HousingReader_AS11_User_Data_128Byte_1[88];
	HwOutputs.HousingReader_AS11_User_Data_128Byte_1[89] := PlcOutputs.HousingReader_AS11_User_Data_128Byte_1[89];
	HwOutputs.HousingReader_AS11_User_Data_128Byte_1[90] := PlcOutputs.HousingReader_AS11_User_Data_128Byte_1[90];
	HwOutputs.HousingReader_AS11_User_Data_128Byte_1[91] := PlcOutputs.HousingReader_AS11_User_Data_128Byte_1[91];
	HwOutputs.HousingReader_AS11_User_Data_128Byte_1[92] := PlcOutputs.HousingReader_AS11_User_Data_128Byte_1[92];
	HwOutputs.HousingReader_AS11_User_Data_128Byte_1[93] := PlcOutputs.HousingReader_AS11_User_Data_128Byte_1[93];
	HwOutputs.HousingReader_AS11_User_Data_128Byte_1[94] := PlcOutputs.HousingReader_AS11_User_Data_128Byte_1[94];
	HwOutputs.HousingReader_AS11_User_Data_128Byte_1[95] := PlcOutputs.HousingReader_AS11_User_Data_128Byte_1[95];
	HwOutputs.HousingReader_AS11_User_Data_128Byte_1[96] := PlcOutputs.HousingReader_AS11_User_Data_128Byte_1[96];
	HwOutputs.HousingReader_AS11_User_Data_128Byte_1[97] := PlcOutputs.HousingReader_AS11_User_Data_128Byte_1[97];
	HwOutputs.HousingReader_AS11_User_Data_128Byte_1[98] := PlcOutputs.HousingReader_AS11_User_Data_128Byte_1[98];
	HwOutputs.HousingReader_AS11_User_Data_128Byte_1[99] := PlcOutputs.HousingReader_AS11_User_Data_128Byte_1[99];
	HwOutputs.HousingReader_AS11_User_Data_128Byte_1[100] := PlcOutputs.HousingReader_AS11_User_Data_128Byte_1[100];
	HwOutputs.HousingReader_AS11_User_Data_128Byte_1[101] := PlcOutputs.HousingReader_AS11_User_Data_128Byte_1[101];
	HwOutputs.HousingReader_AS11_User_Data_128Byte_1[102] := PlcOutputs.HousingReader_AS11_User_Data_128Byte_1[102];
	HwOutputs.HousingReader_AS11_User_Data_128Byte_1[103] := PlcOutputs.HousingReader_AS11_User_Data_128Byte_1[103];
	HwOutputs.HousingReader_AS11_User_Data_128Byte_1[104] := PlcOutputs.HousingReader_AS11_User_Data_128Byte_1[104];
	HwOutputs.HousingReader_AS11_User_Data_128Byte_1[105] := PlcOutputs.HousingReader_AS11_User_Data_128Byte_1[105];
	HwOutputs.HousingReader_AS11_User_Data_128Byte_1[106] := PlcOutputs.HousingReader_AS11_User_Data_128Byte_1[106];
	HwOutputs.HousingReader_AS11_User_Data_128Byte_1[107] := PlcOutputs.HousingReader_AS11_User_Data_128Byte_1[107];
	HwOutputs.HousingReader_AS11_User_Data_128Byte_1[108] := PlcOutputs.HousingReader_AS11_User_Data_128Byte_1[108];
	HwOutputs.HousingReader_AS11_User_Data_128Byte_1[109] := PlcOutputs.HousingReader_AS11_User_Data_128Byte_1[109];
	HwOutputs.HousingReader_AS11_User_Data_128Byte_1[110] := PlcOutputs.HousingReader_AS11_User_Data_128Byte_1[110];
	HwOutputs.HousingReader_AS11_User_Data_128Byte_1[111] := PlcOutputs.HousingReader_AS11_User_Data_128Byte_1[111];
	HwOutputs.HousingReader_AS11_User_Data_128Byte_1[112] := PlcOutputs.HousingReader_AS11_User_Data_128Byte_1[112];
	HwOutputs.HousingReader_AS11_User_Data_128Byte_1[113] := PlcOutputs.HousingReader_AS11_User_Data_128Byte_1[113];
	HwOutputs.HousingReader_AS11_User_Data_128Byte_1[114] := PlcOutputs.HousingReader_AS11_User_Data_128Byte_1[114];
	HwOutputs.HousingReader_AS11_User_Data_128Byte_1[115] := PlcOutputs.HousingReader_AS11_User_Data_128Byte_1[115];
	HwOutputs.HousingReader_AS11_User_Data_128Byte_1[116] := PlcOutputs.HousingReader_AS11_User_Data_128Byte_1[116];
	HwOutputs.HousingReader_AS11_User_Data_128Byte_1[117] := PlcOutputs.HousingReader_AS11_User_Data_128Byte_1[117];
	HwOutputs.HousingReader_AS11_User_Data_128Byte_1[118] := PlcOutputs.HousingReader_AS11_User_Data_128Byte_1[118];
	HwOutputs.HousingReader_AS11_User_Data_128Byte_1[119] := PlcOutputs.HousingReader_AS11_User_Data_128Byte_1[119];
	HwOutputs.HousingReader_AS11_User_Data_128Byte_1[120] := PlcOutputs.HousingReader_AS11_User_Data_128Byte_1[120];
	HwOutputs.HousingReader_AS11_User_Data_128Byte_1[121] := PlcOutputs.HousingReader_AS11_User_Data_128Byte_1[121];
	HwOutputs.HousingReader_AS11_User_Data_128Byte_1[122] := PlcOutputs.HousingReader_AS11_User_Data_128Byte_1[122];
	HwOutputs.HousingReader_AS11_User_Data_128Byte_1[123] := PlcOutputs.HousingReader_AS11_User_Data_128Byte_1[123];
	HwOutputs.HousingReader_AS11_User_Data_128Byte_1[124] := PlcOutputs.HousingReader_AS11_User_Data_128Byte_1[124];
	HwOutputs.HousingReader_AS11_User_Data_128Byte_1[125] := PlcOutputs.HousingReader_AS11_User_Data_128Byte_1[125];
	HwOutputs.HousingReader_AS11_User_Data_128Byte_1[126] := PlcOutputs.HousingReader_AS11_User_Data_128Byte_1[126];
	HwOutputs.HousingReader_AS11_User_Data_128Byte_1[127] := PlcOutputs.HousingReader_AS11_User_Data_128Byte_1[127];
	HwOutputs.HousingReader_AS11_User_Data_128Byte_1[128] := PlcOutputs.HousingReader_AS11_User_Data_128Byte_1[128];
	HwOutputs.HousingReader_AS11_User_Data_128Byte_1[129] := PlcOutputs.HousingReader_AS11_User_Data_128Byte_1[129];
	HwOutputs.CPX_PneuOst_AS10_2_MPA1S_VMPA1_FB_EMS_8_8DO_1 := PlcOutputs.CPX_PneuOst_AS10_2_MPA1S_VMPA1_FB_EMS_8_8DO_1;
	HwOutputs.CPX_PneuOst_AS10_2_MPA1S_VMPA1_FB_EMS_8_8DO_3 := PlcOutputs.CPX_PneuOst_AS10_2_MPA1S_VMPA1_FB_EMS_8_8DO_3;
	HwOutputs.CPX_PneuOst_AS10_2_MPA1S_VMPA1_FB_EMS_8_8DO_2 := PlcOutputs.CPX_PneuOst_AS10_2_MPA1S_VMPA1_FB_EMS_8_8DO_2;
	HwOutputs.CPX_PneuOst_AS10_2_MPA1G_VMPA1_FB_EMG_8_8DO_1 := PlcOutputs.CPX_PneuOst_AS10_2_MPA1G_VMPA1_FB_EMG_8_8DO_1;
	HwOutputs.FlashingReader_Latch_and_Error_Clear_Control_Bits_1 := PlcOutputs.FlashingReader_Latch_and_Error_Clear_Control_Bits_1;
	HwOutputs.FlashingReader_Operation_instruction_Control_Bits_1 := PlcOutputs.FlashingReader_Operation_instruction_Control_Bits_1;
	HwOutputs.FlashingReader_Completion_Clear_Control_Bits_1 := PlcOutputs.FlashingReader_Completion_Clear_Control_Bits_1;
	HwOutputs.FlashingReader_Parameter_Bank_Number_1 := PlcOutputs.FlashingReader_Parameter_Bank_Number_1;
	HwOutputs.FlashingReader_User_Data_128Byte_1[0] := PlcOutputs.FlashingReader_User_Data_128Byte_1[0];
	HwOutputs.FlashingReader_User_Data_128Byte_1[1] := PlcOutputs.FlashingReader_User_Data_128Byte_1[1];
	HwOutputs.FlashingReader_User_Data_128Byte_1[2] := PlcOutputs.FlashingReader_User_Data_128Byte_1[2];
	HwOutputs.FlashingReader_User_Data_128Byte_1[3] := PlcOutputs.FlashingReader_User_Data_128Byte_1[3];
	HwOutputs.FlashingReader_User_Data_128Byte_1[4] := PlcOutputs.FlashingReader_User_Data_128Byte_1[4];
	HwOutputs.FlashingReader_User_Data_128Byte_1[5] := PlcOutputs.FlashingReader_User_Data_128Byte_1[5];
	HwOutputs.FlashingReader_User_Data_128Byte_1[6] := PlcOutputs.FlashingReader_User_Data_128Byte_1[6];
	HwOutputs.FlashingReader_User_Data_128Byte_1[7] := PlcOutputs.FlashingReader_User_Data_128Byte_1[7];
	HwOutputs.FlashingReader_User_Data_128Byte_1[8] := PlcOutputs.FlashingReader_User_Data_128Byte_1[8];
	HwOutputs.FlashingReader_User_Data_128Byte_1[9] := PlcOutputs.FlashingReader_User_Data_128Byte_1[9];
	HwOutputs.FlashingReader_User_Data_128Byte_1[10] := PlcOutputs.FlashingReader_User_Data_128Byte_1[10];
	HwOutputs.FlashingReader_User_Data_128Byte_1[11] := PlcOutputs.FlashingReader_User_Data_128Byte_1[11];
	HwOutputs.FlashingReader_User_Data_128Byte_1[12] := PlcOutputs.FlashingReader_User_Data_128Byte_1[12];
	HwOutputs.FlashingReader_User_Data_128Byte_1[13] := PlcOutputs.FlashingReader_User_Data_128Byte_1[13];
	HwOutputs.FlashingReader_User_Data_128Byte_1[14] := PlcOutputs.FlashingReader_User_Data_128Byte_1[14];
	HwOutputs.FlashingReader_User_Data_128Byte_1[15] := PlcOutputs.FlashingReader_User_Data_128Byte_1[15];
	HwOutputs.FlashingReader_User_Data_128Byte_1[16] := PlcOutputs.FlashingReader_User_Data_128Byte_1[16];
	HwOutputs.FlashingReader_User_Data_128Byte_1[17] := PlcOutputs.FlashingReader_User_Data_128Byte_1[17];
	HwOutputs.FlashingReader_User_Data_128Byte_1[18] := PlcOutputs.FlashingReader_User_Data_128Byte_1[18];
	HwOutputs.FlashingReader_User_Data_128Byte_1[19] := PlcOutputs.FlashingReader_User_Data_128Byte_1[19];
	HwOutputs.FlashingReader_User_Data_128Byte_1[20] := PlcOutputs.FlashingReader_User_Data_128Byte_1[20];
	HwOutputs.FlashingReader_User_Data_128Byte_1[21] := PlcOutputs.FlashingReader_User_Data_128Byte_1[21];
	HwOutputs.FlashingReader_User_Data_128Byte_1[22] := PlcOutputs.FlashingReader_User_Data_128Byte_1[22];
	HwOutputs.FlashingReader_User_Data_128Byte_1[23] := PlcOutputs.FlashingReader_User_Data_128Byte_1[23];
	HwOutputs.FlashingReader_User_Data_128Byte_1[24] := PlcOutputs.FlashingReader_User_Data_128Byte_1[24];
	HwOutputs.FlashingReader_User_Data_128Byte_1[25] := PlcOutputs.FlashingReader_User_Data_128Byte_1[25];
	HwOutputs.FlashingReader_User_Data_128Byte_1[26] := PlcOutputs.FlashingReader_User_Data_128Byte_1[26];
	HwOutputs.FlashingReader_User_Data_128Byte_1[27] := PlcOutputs.FlashingReader_User_Data_128Byte_1[27];
	HwOutputs.FlashingReader_User_Data_128Byte_1[28] := PlcOutputs.FlashingReader_User_Data_128Byte_1[28];
	HwOutputs.FlashingReader_User_Data_128Byte_1[29] := PlcOutputs.FlashingReader_User_Data_128Byte_1[29];
	HwOutputs.FlashingReader_User_Data_128Byte_1[30] := PlcOutputs.FlashingReader_User_Data_128Byte_1[30];
	HwOutputs.FlashingReader_User_Data_128Byte_1[31] := PlcOutputs.FlashingReader_User_Data_128Byte_1[31];
	HwOutputs.FlashingReader_User_Data_128Byte_1[32] := PlcOutputs.FlashingReader_User_Data_128Byte_1[32];
	HwOutputs.FlashingReader_User_Data_128Byte_1[33] := PlcOutputs.FlashingReader_User_Data_128Byte_1[33];
	HwOutputs.FlashingReader_User_Data_128Byte_1[34] := PlcOutputs.FlashingReader_User_Data_128Byte_1[34];
	HwOutputs.FlashingReader_User_Data_128Byte_1[35] := PlcOutputs.FlashingReader_User_Data_128Byte_1[35];
	HwOutputs.FlashingReader_User_Data_128Byte_1[36] := PlcOutputs.FlashingReader_User_Data_128Byte_1[36];
	HwOutputs.FlashingReader_User_Data_128Byte_1[37] := PlcOutputs.FlashingReader_User_Data_128Byte_1[37];
	HwOutputs.FlashingReader_User_Data_128Byte_1[38] := PlcOutputs.FlashingReader_User_Data_128Byte_1[38];
	HwOutputs.FlashingReader_User_Data_128Byte_1[39] := PlcOutputs.FlashingReader_User_Data_128Byte_1[39];
	HwOutputs.FlashingReader_User_Data_128Byte_1[40] := PlcOutputs.FlashingReader_User_Data_128Byte_1[40];
	HwOutputs.FlashingReader_User_Data_128Byte_1[41] := PlcOutputs.FlashingReader_User_Data_128Byte_1[41];
	HwOutputs.FlashingReader_User_Data_128Byte_1[42] := PlcOutputs.FlashingReader_User_Data_128Byte_1[42];
	HwOutputs.FlashingReader_User_Data_128Byte_1[43] := PlcOutputs.FlashingReader_User_Data_128Byte_1[43];
	HwOutputs.FlashingReader_User_Data_128Byte_1[44] := PlcOutputs.FlashingReader_User_Data_128Byte_1[44];
	HwOutputs.FlashingReader_User_Data_128Byte_1[45] := PlcOutputs.FlashingReader_User_Data_128Byte_1[45];
	HwOutputs.FlashingReader_User_Data_128Byte_1[46] := PlcOutputs.FlashingReader_User_Data_128Byte_1[46];
	HwOutputs.FlashingReader_User_Data_128Byte_1[47] := PlcOutputs.FlashingReader_User_Data_128Byte_1[47];
	HwOutputs.FlashingReader_User_Data_128Byte_1[48] := PlcOutputs.FlashingReader_User_Data_128Byte_1[48];
	HwOutputs.FlashingReader_User_Data_128Byte_1[49] := PlcOutputs.FlashingReader_User_Data_128Byte_1[49];
	HwOutputs.FlashingReader_User_Data_128Byte_1[50] := PlcOutputs.FlashingReader_User_Data_128Byte_1[50];
	HwOutputs.FlashingReader_User_Data_128Byte_1[51] := PlcOutputs.FlashingReader_User_Data_128Byte_1[51];
	HwOutputs.FlashingReader_User_Data_128Byte_1[52] := PlcOutputs.FlashingReader_User_Data_128Byte_1[52];
	HwOutputs.FlashingReader_User_Data_128Byte_1[53] := PlcOutputs.FlashingReader_User_Data_128Byte_1[53];
	HwOutputs.FlashingReader_User_Data_128Byte_1[54] := PlcOutputs.FlashingReader_User_Data_128Byte_1[54];
	HwOutputs.FlashingReader_User_Data_128Byte_1[55] := PlcOutputs.FlashingReader_User_Data_128Byte_1[55];
	HwOutputs.FlashingReader_User_Data_128Byte_1[56] := PlcOutputs.FlashingReader_User_Data_128Byte_1[56];
	HwOutputs.FlashingReader_User_Data_128Byte_1[57] := PlcOutputs.FlashingReader_User_Data_128Byte_1[57];
	HwOutputs.FlashingReader_User_Data_128Byte_1[58] := PlcOutputs.FlashingReader_User_Data_128Byte_1[58];
	HwOutputs.FlashingReader_User_Data_128Byte_1[59] := PlcOutputs.FlashingReader_User_Data_128Byte_1[59];
	HwOutputs.FlashingReader_User_Data_128Byte_1[60] := PlcOutputs.FlashingReader_User_Data_128Byte_1[60];
	HwOutputs.FlashingReader_User_Data_128Byte_1[61] := PlcOutputs.FlashingReader_User_Data_128Byte_1[61];
	HwOutputs.FlashingReader_User_Data_128Byte_1[62] := PlcOutputs.FlashingReader_User_Data_128Byte_1[62];
	HwOutputs.FlashingReader_User_Data_128Byte_1[63] := PlcOutputs.FlashingReader_User_Data_128Byte_1[63];
	HwOutputs.FlashingReader_User_Data_128Byte_1[64] := PlcOutputs.FlashingReader_User_Data_128Byte_1[64];
	HwOutputs.FlashingReader_User_Data_128Byte_1[65] := PlcOutputs.FlashingReader_User_Data_128Byte_1[65];
	HwOutputs.FlashingReader_User_Data_128Byte_1[66] := PlcOutputs.FlashingReader_User_Data_128Byte_1[66];
	HwOutputs.FlashingReader_User_Data_128Byte_1[67] := PlcOutputs.FlashingReader_User_Data_128Byte_1[67];
	HwOutputs.FlashingReader_User_Data_128Byte_1[68] := PlcOutputs.FlashingReader_User_Data_128Byte_1[68];
	HwOutputs.FlashingReader_User_Data_128Byte_1[69] := PlcOutputs.FlashingReader_User_Data_128Byte_1[69];
	HwOutputs.FlashingReader_User_Data_128Byte_1[70] := PlcOutputs.FlashingReader_User_Data_128Byte_1[70];
	HwOutputs.FlashingReader_User_Data_128Byte_1[71] := PlcOutputs.FlashingReader_User_Data_128Byte_1[71];
	HwOutputs.FlashingReader_User_Data_128Byte_1[72] := PlcOutputs.FlashingReader_User_Data_128Byte_1[72];
	HwOutputs.FlashingReader_User_Data_128Byte_1[73] := PlcOutputs.FlashingReader_User_Data_128Byte_1[73];
	HwOutputs.FlashingReader_User_Data_128Byte_1[74] := PlcOutputs.FlashingReader_User_Data_128Byte_1[74];
	HwOutputs.FlashingReader_User_Data_128Byte_1[75] := PlcOutputs.FlashingReader_User_Data_128Byte_1[75];
	HwOutputs.FlashingReader_User_Data_128Byte_1[76] := PlcOutputs.FlashingReader_User_Data_128Byte_1[76];
	HwOutputs.FlashingReader_User_Data_128Byte_1[77] := PlcOutputs.FlashingReader_User_Data_128Byte_1[77];
	HwOutputs.FlashingReader_User_Data_128Byte_1[78] := PlcOutputs.FlashingReader_User_Data_128Byte_1[78];
	HwOutputs.FlashingReader_User_Data_128Byte_1[79] := PlcOutputs.FlashingReader_User_Data_128Byte_1[79];
	HwOutputs.FlashingReader_User_Data_128Byte_1[80] := PlcOutputs.FlashingReader_User_Data_128Byte_1[80];
	HwOutputs.FlashingReader_User_Data_128Byte_1[81] := PlcOutputs.FlashingReader_User_Data_128Byte_1[81];
	HwOutputs.FlashingReader_User_Data_128Byte_1[82] := PlcOutputs.FlashingReader_User_Data_128Byte_1[82];
	HwOutputs.FlashingReader_User_Data_128Byte_1[83] := PlcOutputs.FlashingReader_User_Data_128Byte_1[83];
	HwOutputs.FlashingReader_User_Data_128Byte_1[84] := PlcOutputs.FlashingReader_User_Data_128Byte_1[84];
	HwOutputs.FlashingReader_User_Data_128Byte_1[85] := PlcOutputs.FlashingReader_User_Data_128Byte_1[85];
	HwOutputs.FlashingReader_User_Data_128Byte_1[86] := PlcOutputs.FlashingReader_User_Data_128Byte_1[86];
	HwOutputs.FlashingReader_User_Data_128Byte_1[87] := PlcOutputs.FlashingReader_User_Data_128Byte_1[87];
	HwOutputs.FlashingReader_User_Data_128Byte_1[88] := PlcOutputs.FlashingReader_User_Data_128Byte_1[88];
	HwOutputs.FlashingReader_User_Data_128Byte_1[89] := PlcOutputs.FlashingReader_User_Data_128Byte_1[89];
	HwOutputs.FlashingReader_User_Data_128Byte_1[90] := PlcOutputs.FlashingReader_User_Data_128Byte_1[90];
	HwOutputs.FlashingReader_User_Data_128Byte_1[91] := PlcOutputs.FlashingReader_User_Data_128Byte_1[91];
	HwOutputs.FlashingReader_User_Data_128Byte_1[92] := PlcOutputs.FlashingReader_User_Data_128Byte_1[92];
	HwOutputs.FlashingReader_User_Data_128Byte_1[93] := PlcOutputs.FlashingReader_User_Data_128Byte_1[93];
	HwOutputs.FlashingReader_User_Data_128Byte_1[94] := PlcOutputs.FlashingReader_User_Data_128Byte_1[94];
	HwOutputs.FlashingReader_User_Data_128Byte_1[95] := PlcOutputs.FlashingReader_User_Data_128Byte_1[95];
	HwOutputs.FlashingReader_User_Data_128Byte_1[96] := PlcOutputs.FlashingReader_User_Data_128Byte_1[96];
	HwOutputs.FlashingReader_User_Data_128Byte_1[97] := PlcOutputs.FlashingReader_User_Data_128Byte_1[97];
	HwOutputs.FlashingReader_User_Data_128Byte_1[98] := PlcOutputs.FlashingReader_User_Data_128Byte_1[98];
	HwOutputs.FlashingReader_User_Data_128Byte_1[99] := PlcOutputs.FlashingReader_User_Data_128Byte_1[99];
	HwOutputs.FlashingReader_User_Data_128Byte_1[100] := PlcOutputs.FlashingReader_User_Data_128Byte_1[100];
	HwOutputs.FlashingReader_User_Data_128Byte_1[101] := PlcOutputs.FlashingReader_User_Data_128Byte_1[101];
	HwOutputs.FlashingReader_User_Data_128Byte_1[102] := PlcOutputs.FlashingReader_User_Data_128Byte_1[102];
	HwOutputs.FlashingReader_User_Data_128Byte_1[103] := PlcOutputs.FlashingReader_User_Data_128Byte_1[103];
	HwOutputs.FlashingReader_User_Data_128Byte_1[104] := PlcOutputs.FlashingReader_User_Data_128Byte_1[104];
	HwOutputs.FlashingReader_User_Data_128Byte_1[105] := PlcOutputs.FlashingReader_User_Data_128Byte_1[105];
	HwOutputs.FlashingReader_User_Data_128Byte_1[106] := PlcOutputs.FlashingReader_User_Data_128Byte_1[106];
	HwOutputs.FlashingReader_User_Data_128Byte_1[107] := PlcOutputs.FlashingReader_User_Data_128Byte_1[107];
	HwOutputs.FlashingReader_User_Data_128Byte_1[108] := PlcOutputs.FlashingReader_User_Data_128Byte_1[108];
	HwOutputs.FlashingReader_User_Data_128Byte_1[109] := PlcOutputs.FlashingReader_User_Data_128Byte_1[109];
	HwOutputs.FlashingReader_User_Data_128Byte_1[110] := PlcOutputs.FlashingReader_User_Data_128Byte_1[110];
	HwOutputs.FlashingReader_User_Data_128Byte_1[111] := PlcOutputs.FlashingReader_User_Data_128Byte_1[111];
	HwOutputs.FlashingReader_User_Data_128Byte_1[112] := PlcOutputs.FlashingReader_User_Data_128Byte_1[112];
	HwOutputs.FlashingReader_User_Data_128Byte_1[113] := PlcOutputs.FlashingReader_User_Data_128Byte_1[113];
	HwOutputs.FlashingReader_User_Data_128Byte_1[114] := PlcOutputs.FlashingReader_User_Data_128Byte_1[114];
	HwOutputs.FlashingReader_User_Data_128Byte_1[115] := PlcOutputs.FlashingReader_User_Data_128Byte_1[115];
	HwOutputs.FlashingReader_User_Data_128Byte_1[116] := PlcOutputs.FlashingReader_User_Data_128Byte_1[116];
	HwOutputs.FlashingReader_User_Data_128Byte_1[117] := PlcOutputs.FlashingReader_User_Data_128Byte_1[117];
	HwOutputs.FlashingReader_User_Data_128Byte_1[118] := PlcOutputs.FlashingReader_User_Data_128Byte_1[118];
	HwOutputs.FlashingReader_User_Data_128Byte_1[119] := PlcOutputs.FlashingReader_User_Data_128Byte_1[119];
	HwOutputs.FlashingReader_User_Data_128Byte_1[120] := PlcOutputs.FlashingReader_User_Data_128Byte_1[120];
	HwOutputs.FlashingReader_User_Data_128Byte_1[121] := PlcOutputs.FlashingReader_User_Data_128Byte_1[121];
	HwOutputs.FlashingReader_User_Data_128Byte_1[122] := PlcOutputs.FlashingReader_User_Data_128Byte_1[122];
	HwOutputs.FlashingReader_User_Data_128Byte_1[123] := PlcOutputs.FlashingReader_User_Data_128Byte_1[123];
	HwOutputs.FlashingReader_User_Data_128Byte_1[124] := PlcOutputs.FlashingReader_User_Data_128Byte_1[124];
	HwOutputs.FlashingReader_User_Data_128Byte_1[125] := PlcOutputs.FlashingReader_User_Data_128Byte_1[125];
	HwOutputs.FlashingReader_User_Data_128Byte_1[126] := PlcOutputs.FlashingReader_User_Data_128Byte_1[126];
	HwOutputs.FlashingReader_User_Data_128Byte_1[127] := PlcOutputs.FlashingReader_User_Data_128Byte_1[127];
	HwOutputs.FlashingReader_User_Data_128Byte_1[128] := PlcOutputs.FlashingReader_User_Data_128Byte_1[128];
	HwOutputs.FlashingReader_User_Data_128Byte_1[129] := PlcOutputs.FlashingReader_User_Data_128Byte_1[129];
	HwOutputs.AS10_2flashing_Out_64_Byte_1[0] := PlcOutputs.AS10_2flashing_Out_64_Byte_1[0];
	HwOutputs.AS10_2flashing_Out_64_Byte_1[1] := PlcOutputs.AS10_2flashing_Out_64_Byte_1[1];
	HwOutputs.AS10_2flashing_Out_64_Byte_1[2] := PlcOutputs.AS10_2flashing_Out_64_Byte_1[2];
	HwOutputs.AS10_2flashing_Out_64_Byte_1[3] := PlcOutputs.AS10_2flashing_Out_64_Byte_1[3];
	HwOutputs.AS10_2flashing_Out_64_Byte_1[4] := PlcOutputs.AS10_2flashing_Out_64_Byte_1[4];
	HwOutputs.AS10_2flashing_Out_64_Byte_1[5] := PlcOutputs.AS10_2flashing_Out_64_Byte_1[5];
	HwOutputs.AS10_2flashing_Out_64_Byte_1[6] := PlcOutputs.AS10_2flashing_Out_64_Byte_1[6];
	HwOutputs.AS10_2flashing_Out_64_Byte_1[7] := PlcOutputs.AS10_2flashing_Out_64_Byte_1[7];
	HwOutputs.AS10_2flashing_Out_64_Byte_1[8] := PlcOutputs.AS10_2flashing_Out_64_Byte_1[8];
	HwOutputs.AS10_2flashing_Out_64_Byte_1[9] := PlcOutputs.AS10_2flashing_Out_64_Byte_1[9];
	HwOutputs.AS10_2flashing_Out_64_Byte_1[10] := PlcOutputs.AS10_2flashing_Out_64_Byte_1[10];
	HwOutputs.AS10_2flashing_Out_64_Byte_1[11] := PlcOutputs.AS10_2flashing_Out_64_Byte_1[11];
	HwOutputs.AS10_2flashing_Out_64_Byte_1[12] := PlcOutputs.AS10_2flashing_Out_64_Byte_1[12];
	HwOutputs.AS10_2flashing_Out_64_Byte_1[13] := PlcOutputs.AS10_2flashing_Out_64_Byte_1[13];
	HwOutputs.AS10_2flashing_Out_64_Byte_1[14] := PlcOutputs.AS10_2flashing_Out_64_Byte_1[14];
	HwOutputs.AS10_2flashing_Out_64_Byte_1[15] := PlcOutputs.AS10_2flashing_Out_64_Byte_1[15];
	HwOutputs.AS10_2flashing_Out_64_Byte_1[16] := PlcOutputs.AS10_2flashing_Out_64_Byte_1[16];
	HwOutputs.AS10_2flashing_Out_64_Byte_1[17] := PlcOutputs.AS10_2flashing_Out_64_Byte_1[17];
	HwOutputs.AS10_2flashing_Out_64_Byte_1[18] := PlcOutputs.AS10_2flashing_Out_64_Byte_1[18];
	HwOutputs.AS10_2flashing_Out_64_Byte_1[19] := PlcOutputs.AS10_2flashing_Out_64_Byte_1[19];
	HwOutputs.AS10_2flashing_Out_64_Byte_1[20] := PlcOutputs.AS10_2flashing_Out_64_Byte_1[20];
	HwOutputs.AS10_2flashing_Out_64_Byte_1[21] := PlcOutputs.AS10_2flashing_Out_64_Byte_1[21];
	HwOutputs.AS10_2flashing_Out_64_Byte_1[22] := PlcOutputs.AS10_2flashing_Out_64_Byte_1[22];
	HwOutputs.AS10_2flashing_Out_64_Byte_1[23] := PlcOutputs.AS10_2flashing_Out_64_Byte_1[23];
	HwOutputs.AS10_2flashing_Out_64_Byte_1[24] := PlcOutputs.AS10_2flashing_Out_64_Byte_1[24];
	HwOutputs.AS10_2flashing_Out_64_Byte_1[25] := PlcOutputs.AS10_2flashing_Out_64_Byte_1[25];
	HwOutputs.AS10_2flashing_Out_64_Byte_1[26] := PlcOutputs.AS10_2flashing_Out_64_Byte_1[26];
	HwOutputs.AS10_2flashing_Out_64_Byte_1[27] := PlcOutputs.AS10_2flashing_Out_64_Byte_1[27];
	HwOutputs.AS10_2flashing_Out_64_Byte_1[28] := PlcOutputs.AS10_2flashing_Out_64_Byte_1[28];
	HwOutputs.AS10_2flashing_Out_64_Byte_1[29] := PlcOutputs.AS10_2flashing_Out_64_Byte_1[29];
	HwOutputs.AS10_2flashing_Out_64_Byte_1[30] := PlcOutputs.AS10_2flashing_Out_64_Byte_1[30];
	HwOutputs.AS10_2flashing_Out_64_Byte_1[31] := PlcOutputs.AS10_2flashing_Out_64_Byte_1[31];
	HwOutputs.AS10_2flashing_Out_64_Byte_1[32] := PlcOutputs.AS10_2flashing_Out_64_Byte_1[32];
	HwOutputs.AS10_2flashing_Out_64_Byte_1[33] := PlcOutputs.AS10_2flashing_Out_64_Byte_1[33];
	HwOutputs.AS10_2flashing_Out_64_Byte_1[34] := PlcOutputs.AS10_2flashing_Out_64_Byte_1[34];
	HwOutputs.AS10_2flashing_Out_64_Byte_1[35] := PlcOutputs.AS10_2flashing_Out_64_Byte_1[35];
	HwOutputs.AS10_2flashing_Out_64_Byte_1[36] := PlcOutputs.AS10_2flashing_Out_64_Byte_1[36];
	HwOutputs.AS10_2flashing_Out_64_Byte_1[37] := PlcOutputs.AS10_2flashing_Out_64_Byte_1[37];
	HwOutputs.AS10_2flashing_Out_64_Byte_1[38] := PlcOutputs.AS10_2flashing_Out_64_Byte_1[38];
	HwOutputs.AS10_2flashing_Out_64_Byte_1[39] := PlcOutputs.AS10_2flashing_Out_64_Byte_1[39];
	HwOutputs.AS10_2flashing_Out_64_Byte_1[40] := PlcOutputs.AS10_2flashing_Out_64_Byte_1[40];
	HwOutputs.AS10_2flashing_Out_64_Byte_1[41] := PlcOutputs.AS10_2flashing_Out_64_Byte_1[41];
	HwOutputs.AS10_2flashing_Out_64_Byte_1[42] := PlcOutputs.AS10_2flashing_Out_64_Byte_1[42];
	HwOutputs.AS10_2flashing_Out_64_Byte_1[43] := PlcOutputs.AS10_2flashing_Out_64_Byte_1[43];
	HwOutputs.AS10_2flashing_Out_64_Byte_1[44] := PlcOutputs.AS10_2flashing_Out_64_Byte_1[44];
	HwOutputs.AS10_2flashing_Out_64_Byte_1[45] := PlcOutputs.AS10_2flashing_Out_64_Byte_1[45];
	HwOutputs.AS10_2flashing_Out_64_Byte_1[46] := PlcOutputs.AS10_2flashing_Out_64_Byte_1[46];
	HwOutputs.AS10_2flashing_Out_64_Byte_1[47] := PlcOutputs.AS10_2flashing_Out_64_Byte_1[47];
	HwOutputs.AS10_2flashing_Out_64_Byte_1[48] := PlcOutputs.AS10_2flashing_Out_64_Byte_1[48];
	HwOutputs.AS10_2flashing_Out_64_Byte_1[49] := PlcOutputs.AS10_2flashing_Out_64_Byte_1[49];
	HwOutputs.AS10_2flashing_Out_64_Byte_1[50] := PlcOutputs.AS10_2flashing_Out_64_Byte_1[50];
	HwOutputs.AS10_2flashing_Out_64_Byte_1[51] := PlcOutputs.AS10_2flashing_Out_64_Byte_1[51];
	HwOutputs.AS10_2flashing_Out_64_Byte_1[52] := PlcOutputs.AS10_2flashing_Out_64_Byte_1[52];
	HwOutputs.AS10_2flashing_Out_64_Byte_1[53] := PlcOutputs.AS10_2flashing_Out_64_Byte_1[53];
	HwOutputs.AS10_2flashing_Out_64_Byte_1[54] := PlcOutputs.AS10_2flashing_Out_64_Byte_1[54];
	HwOutputs.AS10_2flashing_Out_64_Byte_1[55] := PlcOutputs.AS10_2flashing_Out_64_Byte_1[55];
	HwOutputs.AS10_2flashing_Out_64_Byte_1[56] := PlcOutputs.AS10_2flashing_Out_64_Byte_1[56];
	HwOutputs.AS10_2flashing_Out_64_Byte_1[57] := PlcOutputs.AS10_2flashing_Out_64_Byte_1[57];
	HwOutputs.AS10_2flashing_Out_64_Byte_1[58] := PlcOutputs.AS10_2flashing_Out_64_Byte_1[58];
	HwOutputs.AS10_2flashing_Out_64_Byte_1[59] := PlcOutputs.AS10_2flashing_Out_64_Byte_1[59];
	HwOutputs.AS10_2flashing_Out_64_Byte_1[60] := PlcOutputs.AS10_2flashing_Out_64_Byte_1[60];
	HwOutputs.AS10_2flashing_Out_64_Byte_1[61] := PlcOutputs.AS10_2flashing_Out_64_Byte_1[61];
	HwOutputs.AS10_2flashing_Out_64_Byte_1[62] := PlcOutputs.AS10_2flashing_Out_64_Byte_1[62];
	HwOutputs.AS10_2flashing_Out_64_Byte_1[63] := PlcOutputs.AS10_2flashing_Out_64_Byte_1[63];
END_FUNCTION
